		T_Visu.ptrT_ExchgParam^.T_InfoValueCommon.iTotalCountDownCycle:=T_NovRAM.T_Data.T_ProcessImageData.T_AutoGeometryPara.iCycleGeometry;
		T_Visu.ptrT_ExchgParam^.T_InfoValueCommon.iTotalCountDownPlungeCycle:=T_Station.T_WorkTool.iTotalCountDownPlungeCycle;
		T_Visu.ptrT_ExchgParam^.T_InfoValueCommon.iTotalCountDownGrooveCycle:=T_NovRAM.T_Data.T_ProcessImageData.T_AutoGroovePara.iNumberOfGrooves;
		T_Visu.ptrT_ExchgParam^.T_InfoValueCommon.rToolDiameter:=T_NovRAM.T_Data.T_ProcessImageData.T_ProcessPara.rToolDiameterProcess;
		T_Visu.ptrT_ExchgParam^.T_InfoValueCommon.rToolTotalLength:=rToolTotalLength * 10.0;	(* umwandeln von cm in mm *)
		IF (T_Visu.T_PlcParam.dwActualPage = 10) THEN
			IF T_NovRAM.T_Data.T_ProcessImageData.T_AutoGeometryPara.xPlungeActivationGeometry THEN
				T_Visu.ptrT_ExchgParam^.T_InfoValueCommon.rToolTotalLength:=T_Visu.ptrT_ExchgParam^.T_InfoValueCommon.rToolTotalLength + T_NovRAM.T_Data.T_ProcessImageData.T_AutoGeometryPara.rPlungeLengthToolFeedGeometry;
			END_IF;
			IF T_NovRAM.T_Data.T_ProcessImageData.T_AutoGeometryPara.xDisplaceActivationGeometry THEN
				T_Visu.ptrT_ExchgParam^.T_InfoValueCommon.rToolTotalLength:=T_Visu.ptrT_ExchgParam^.T_InfoValueCommon.rToolTotalLength + T_NovRAM.T_Data.T_ProcessImageData.T_AutoGeometryPara.rDisplaceLengthToolFeedGeometry;
			END_IF;
		END_IF;
		IF (T_Visu.T_PlcParam.dwActualPage = 20) THEN
			IF T_NovRAM.T_Data.T_ProcessImageData.T_AutoGroovePara.xPlungeActivationGroove AND NOT(T_NovRAM.T_Data.T_ProcessImageData.T_AutoGroovePara.xBlockGrindFeeder) THEN
				T_Visu.ptrT_ExchgParam^.T_InfoValueCommon.rToolTotalLength:=T_Visu.ptrT_ExchgParam^.T_InfoValueCommon.rToolTotalLength + T_NovRAM.T_Data.T_ProcessImageData.T_AutoGroovePara.rPlungeLengthToolFeedGroove;
			END_IF;
			IF T_NovRAM.T_Data.T_ProcessImageData.T_AutoGroovePara.xDisplaceActivationGroove THEN
				T_Visu.ptrT_ExchgParam^.T_InfoValueCommon.rToolTotalLength:=T_Visu.ptrT_ExchgParam^.T_InfoValueCommon.rToolTotalLength + T_NovRAM.T_Data.T_ProcessImageData.T_AutoGroovePara.rDisplaceLengthToolFeedGroove;
			END_IF;
		END_IF;
	ELSE
		T_Visu.ptrT_ExchgParam^.T_InfoValueCommon.iCountDownCycle:=1;
		T_Visu.ptrT_ExchgParam^.T_InfoValueCommon.iCountDownPlungeCycle:=1;
		T_Visu.ptrT_ExchgParam^.T_InfoValueCommon.iCountDownGrooveCycle:=1;
	END_IF;

(* Tool Geometry Managment *)
	IF (T_Visu.T_PlcParam.dwActualPage = 120) OR (T_Visu.T_PlcParam.dwActualPage = 121) THEN
		FailingEdgeGeometryManagement(CLK:=TRUE);
		RisingEdgeGeometryManagement(CLK:=(T_Visu.T_PlcParam.dwActualPage = 120) OR (T_Visu.T_PlcParam.dwActualPage = 121));
		IF RisingEdgeGeometryManagement.Q THEN
			arSaveToolGeometry:=T_Visu.ptrT_ExchgParam^.T_GeometryCommon.T_Geometry;
		END_IF;
		T_Visu.ptrT_ExchgParam^.T_GeometryCommon.rMinToolDiameter:=T_Visu.ptrT_ExchgParam^.T_StationCommon.T_PrismPara.rToolDiameterMin;
		T_Visu.ptrT_ExchgParam^.T_GeometryCommon.rMaxToolDiameter:=T_Visu.ptrT_ExchgParam^.T_StationCommon.T_PrismPara.rToolDiameterMax;
		T_Visu.ptrT_ExchgParam^.T_GeometryCommon.rMinToolLength:=0.1;
		T_Visu.ptrT_ExchgParam^.T_GeometryCommon.rMaxToolLength:=T_Visu.ptrT_ExchgParam^.T_StationCommon.rConfigMaxToolLength;

		IF (arSaveToolGeometry.arEndDiameter[1] <> T_Visu.ptrT_ExchgParam^.T_GeometryCommon.T_Geometry.arEndDiameter[1]) THEN
			arSaveToolGeometry.arEndDiameter[1]:=T_Visu.ptrT_ExchgParam^.T_GeometryCommon.T_Geometry.arEndDiameter[1];
			arSaveToolGeometry.arStartDiameter[2]:=arSaveToolGeometry.arEndDiameter[1];
			T_Visu.ptrT_ExchgParam^.T_GeometryCommon.T_Geometry.arStartDiameter[2]:=arSaveToolGeometry.arStartDiameter[2];
		END_IF;
		IF (arSaveToolGeometry.arStartDiameter[2] <> T_Visu.ptrT_ExchgParam^.T_GeometryCommon.T_Geometry.arStartDiameter[2]) THEN
			arSaveToolGeometry.arStartDiameter[2]:=T_Visu.ptrT_ExchgParam^.T_GeometryCommon.T_Geometry.arStartDiameter[2];
			arSaveToolGeometry.arEndDiameter[1]:=arSaveToolGeometry.arStartDiameter[2];
			T_Visu.ptrT_ExchgParam^.T_GeometryCommon.T_Geometry.arEndDiameter[1]:=arSaveToolGeometry.arEndDiameter[1];
		END_IF;
		IF (arSaveToolGeometry.arEndDiameter[2] <> T_Visu.ptrT_ExchgParam^.T_GeometryCommon.T_Geometry.arEndDiameter[2]) THEN
			arSaveToolGeometry.arEndDiameter[2]:=T_Visu.ptrT_ExchgParam^.T_GeometryCommon.T_Geometry.arEndDiameter[2];
			arSaveToolGeometry.arStartDiameter[3]:=arSaveToolGeometry.arEndDiameter[2];
			T_Visu.ptrT_ExchgParam^.T_GeometryCommon.T_Geometry.arStartDiameter[3]:=arSaveToolGeometry.arStartDiameter[3];
		END_IF;
		IF (arSaveToolGeometry.arStartDiameter[3] <> T_Visu.ptrT_ExchgParam^.T_GeometryCommon.T_Geometry.arStartDiameter[3]) THEN
			arSaveToolGeometry.arStartDiameter[3]:=T_Visu.ptrT_ExchgParam^.T_GeometryCommon.T_Geometry.arStartDiameter[3];
			arSaveToolGeometry.arEndDiameter[2]:=arSaveToolGeometry.arStartDiameter[3];
			T_Visu.ptrT_ExchgParam^.T_GeometryCommon.T_Geometry.arEndDiameter[2]:=arSaveToolGeometry.arEndDiameter[2];
		END_IF;
		IF (arSaveToolGeometry.arEndDiameter[3] <> T_Visu.ptrT_ExchgParam^.T_GeometryCommon.T_Geometry.arEndDiameter[3]) THEN
			arSaveToolGeometry.arEndDiameter[3]:=T_Visu.ptrT_ExchgParam^.T_GeometryCommon.T_Geometry.arEndDiameter[3];
			arSaveToolGeometry.arStartDiameter[4]:=arSaveToolGeometry.arEndDiameter[3];
			T_Visu.ptrT_ExchgParam^.T_GeometryCommon.T_Geometry.arStartDiameter[4]:=arSaveToolGeometry.arStartDiameter[4];
		END_IF;
		IF (arSaveToolGeometry.arStartDiameter[4] <> T_Visu.ptrT_ExchgParam^.T_GeometryCommon.T_Geometry.arStartDiameter[4]) THEN
			arSaveToolGeometry.arStartDiameter[4]:=T_Visu.ptrT_ExchgParam^.T_GeometryCommon.T_Geometry.arStartDiameter[4];
			arSaveToolGeometry.arEndDiameter[3]:=arSaveToolGeometry.arStartDiameter[4];
			T_Visu.ptrT_ExchgParam^.T_GeometryCommon.T_Geometry.arEndDiameter[3]:=arSaveToolGeometry.arEndDiameter[3];
		END_IF;
(*09.12.2022: SOA	{	 *)
		IF (arSaveToolGeometry.arEndDiameter[4] <> T_Visu.ptrT_ExchgParam^.T_GeometryCommon.T_Geometry.arEndDiameter[4]) THEN
			arSaveToolGeometry.arEndDiameter[4]:=T_Visu.ptrT_ExchgParam^.T_GeometryCommon.T_Geometry.arEndDiameter[4];
			arSaveToolGeometry.arStartDiameter[5]:=arSaveToolGeometry.arEndDiameter[4];
			T_Visu.ptrT_ExchgParam^.T_GeometryCommon.T_Geometry.arStartDiameter[5]:=arSaveToolGeometry.arStartDiameter[5];
		END_IF;
		IF (arSaveToolGeometry.arStartDiameter[5] <> T_Visu.ptrT_ExchgParam^.T_GeometryCommon.T_Geometry.arStartDiameter[5]) THEN
			arSaveToolGeometry.arStartDiameter[5]:=T_Visu.ptrT_ExchgParam^.T_GeometryCommon.T_Geometry.arStartDiameter[5];
			arSaveToolGeometry.arEndDiameter[4]:=arSaveToolGeometry.arStartDiameter[5];
			T_Visu.ptrT_ExchgParam^.T_GeometryCommon.T_Geometry.arEndDiameter[4]:=arSaveToolGeometry.arEndDiameter[4];
		END_IF;
		IF (arSaveToolGeometry.arEndDiameter[5] <> T_Visu.ptrT_ExchgParam^.T_GeometryCommon.T_Geometry.arEndDiameter[5]) THEN
			arSaveToolGeometry.arEndDiameter[5]:=T_Visu.ptrT_ExchgParam^.T_GeometryCommon.T_Geometry.arEndDiameter[5];
			arSaveToolGeometry.arStartDiameter[6]:=arSaveToolGeometry.arEndDiameter[5];
			T_Visu.ptrT_ExchgParam^.T_GeometryCommon.T_Geometry.arStartDiameter[6]:=arSaveToolGeometry.arStartDiameter[6];
		END_IF;
		IF (arSaveToolGeometry.arStartDiameter[6] <> T_Visu.ptrT_ExchgParam^.T_GeometryCommon.T_Geometry.arStartDiameter[6]) THEN
			arSaveToolGeometry.arStartDiameter[6]:=T_Visu.ptrT_ExchgParam^.T_GeometryCommon.T_Geometry.arStartDiameter[6];
			arSaveToolGeometry.arEndDiameter[5]:=arSaveToolGeometry.arStartDiameter[6];
			T_Visu.ptrT_ExchgParam^.T_GeometryCommon.T_Geometry.arEndDiameter[5]:=arSaveToolGeometry.arEndDiameter[5];
		END_IF;
(*09.12.2022: SOA	}	 *)

(*Select Form*)
		FOR ii:=1 TO 6 DO
			IF NOT(T_Visu.ptrT_ExchgParam^.T_GeometryCommon.T_Geometry.axActiveSection[ii]) THEN
				T_Visu.ptrT_ExchgParam^.T_GeometryCommon.abSectionSelectForm[ii]:=0;
			END_IF;
		END_FOR;
		FOR ii:=1 TO 6 DO
			IF (T_Visu.ptrT_ExchgParam^.T_GeometryCommon.T_Geometry.arStartDiameter[ii] = T_Visu.ptrT_ExchgParam^.T_GeometryCommon.T_Geometry.arEndDiameter[ii]) THEN
				IF T_Visu.ptrT_ExchgParam^.T_GeometryCommon.T_Geometry.axActiveSection[ii] THEN
					T_Visu.ptrT_ExchgParam^.T_GeometryCommon.abSectionSelectForm[ii]:=2;
				END_IF;
			END_IF;
		END_FOR;
		FOR ii:=1 TO 6 DO
			IF (T_Visu.ptrT_ExchgParam^.T_GeometryCommon.T_Geometry.arStartDiameter[ii] > T_Visu.ptrT_ExchgParam^.T_GeometryCommon.T_Geometry.arEndDiameter[ii]) THEN
				IF T_Visu.ptrT_ExchgParam^.T_GeometryCommon.T_Geometry.axActiveSection[ii] THEN
					T_Visu.ptrT_ExchgParam^.T_GeometryCommon.abSectionSelectForm[ii]:=3;
				END_IF;
			END_IF;
		END_FOR;
		FOR ii:=1 TO 6 DO
			IF (T_Visu.ptrT_ExchgParam^.T_GeometryCommon.T_Geometry.arStartDiameter[ii] < T_Visu.ptrT_ExchgParam^.T_GeometryCommon.T_Geometry.arEndDiameter[ii]) THEN
				IF T_Visu.ptrT_ExchgParam^.T_GeometryCommon.T_Geometry.axActiveSection[ii] THEN
					T_Visu.ptrT_ExchgParam^.T_GeometryCommon.abSectionSelectForm[ii]:=4;
				END_IF;
			END_IF;
		END_FOR;

 (*Checking for forbidden ToolDiameter - if forbidden: Set Bit in Word *)
	rCalcTotalToolLength:=0.0;
		FOR ii:=1 TO 6 DO
			IF ii>=1 AND ii<=4 THEN
				IF (T_Visu.ptrT_ExchgParam^.T_GeometryCommon.T_Geometry.arStartDiameter[ii] = 0) OR
				     (T_Visu.ptrT_ExchgParam^.T_GeometryCommon.T_Geometry.arStartDiameter[ii] > T_Visu.ptrT_ExchgParam^.T_StationCommon.T_PrismPara.rToolDiameterMax) OR
				     (T_Visu.ptrT_ExchgParam^.T_GeometryCommon.T_Geometry.arStartDiameter[ii] < T_Visu.ptrT_ExchgParam^.T_StationCommon.T_PrismPara.rToolDiameterMin) THEN
					T_Visu.ptrT_ExchgParam^.T_GeometryCommon.wWrongInput:=DWORD_TO_WORD(SETBIT32(T_Visu.ptrT_ExchgParam^.T_GeometryCommon.wWrongInput,INT_TO_SINT(ii-1)));
				ELSE
					T_Visu.ptrT_ExchgParam^.T_GeometryCommon.wWrongInput:=DWORD_TO_WORD(CLEARBIT32(T_Visu.ptrT_ExchgParam^.T_GeometryCommon.wWrongInput,INT_TO_SINT(ii-1)));
				END_IF;
				IF (T_Visu.ptrT_ExchgParam^.T_GeometryCommon.T_Geometry.arEndDiameter[ii] = 0) OR
				     (T_Visu.ptrT_ExchgParam^.T_GeometryCommon.T_Geometry.arEndDiameter[ii] > T_Visu.ptrT_ExchgParam^.T_StationCommon.T_PrismPara.rToolDiameterMax) OR
				     (T_Visu.ptrT_ExchgParam^.T_GeometryCommon.T_Geometry.arEndDiameter[ii] < T_Visu.ptrT_ExchgParam^.T_StationCommon.T_PrismPara.rToolDiameterMin) THEN
					T_Visu.ptrT_ExchgParam^.T_GeometryCommon.wWrongInput:=DWORD_TO_WORD(SETBIT32(T_Visu.ptrT_ExchgParam^.T_GeometryCommon.wWrongInput,INT_TO_SINT(ii+3)));
				ELSE
					T_Visu.ptrT_ExchgParam^.T_GeometryCommon.wWrongInput:=DWORD_TO_WORD(CLEARBIT32(T_Visu.ptrT_ExchgParam^.T_GeometryCommon.wWrongInput,INT_TO_SINT(ii+3)));
				END_IF;
				IF (T_Visu.ptrT_ExchgParam^.T_GeometryCommon.T_Geometry.arSectionPitch[ii] = 0) THEN
					T_Visu.ptrT_ExchgParam^.T_GeometryCommon.wWrongInput:=DWORD_TO_WORD(SETBIT32(T_Visu.ptrT_ExchgParam^.T_GeometryCommon.wWrongInput,INT_TO_SINT(ii+7)));
				ELSE
					T_Visu.ptrT_ExchgParam^.T_GeometryCommon.wWrongInput:=DWORD_TO_WORD(CLEARBIT32(T_Visu.ptrT_ExchgParam^.T_GeometryCommon.wWrongInput,INT_TO_SINT(ii+7)));
				END_IF;
				IF (T_Visu.ptrT_ExchgParam^.T_GeometryCommon.T_Geometry.arSectionLength[ii] = 0) THEN
					T_Visu.ptrT_ExchgParam^.T_GeometryCommon.wWrongInput:=DWORD_TO_WORD(SETBIT32(T_Visu.ptrT_ExchgParam^.T_GeometryCommon.wWrongInput,INT_TO_SINT(ii+11)));
				ELSE
					T_Visu.ptrT_ExchgParam^.T_GeometryCommon.wWrongInput:=DWORD_TO_WORD(CLEARBIT32(T_Visu.ptrT_ExchgParam^.T_GeometryCommon.wWrongInput,INT_TO_SINT(ii+11)));
				END_IF;
 (*09.12.2022: SOA *) (*Definition of second variable = wWrongInput_2*)
			ELSIF  ii>=5 AND ii<=6 THEN
				IF (T_Visu.ptrT_ExchgParam^.T_GeometryCommon.T_Geometry.arSectionPitch[ii] = 0) THEN
					T_Visu.ptrT_ExchgParam^.T_GeometryCommon.wWrongInput_2:=DWORD_TO_WORD(SETBIT32(T_Visu.ptrT_ExchgParam^.T_GeometryCommon.wWrongInput_2,INT_TO_SINT(ii-5)));
				ELSE
					T_Visu.ptrT_ExchgParam^.T_GeometryCommon.wWrongInput_2:=DWORD_TO_WORD(CLEARBIT32(T_Visu.ptrT_ExchgParam^.T_GeometryCommon.wWrongInput_2,INT_TO_SINT(ii-5)));
				END_IF;
				IF (T_Visu.ptrT_ExchgParam^.T_GeometryCommon.T_Geometry.arSectionLength[ii] = 0) THEN
					T_Visu.ptrT_ExchgParam^.T_GeometryCommon.wWrongInput_2:=DWORD_TO_WORD(SETBIT32(T_Visu.ptrT_ExchgParam^.T_GeometryCommon.wWrongInput_2,INT_TO_SINT(ii-1)));
				ELSE
					T_Visu.ptrT_ExchgParam^.T_GeometryCommon.wWrongInput_2:=DWORD_TO_WORD(CLEARBIT32(T_Visu.ptrT_ExchgParam^.T_GeometryCommon.wWrongInput_2,INT_TO_SINT(ii-1)));
				END_IF;
			END_IF;

			IF T_Visu.ptrT_ExchgParam^.T_GeometryCommon.T_Geometry.axActiveSection[ii] THEN
				rCalcTotalToolLength:=rCalcTotalToolLength + T_Visu.ptrT_ExchgParam^.T_GeometryCommon.T_Geometry.arSectionLength[ii];
			END_IF;
		END_FOR;

 (*Checking  every Section for active Bits, changing "SelectForm" if active *)
		IF (rCalcTotalToolLength > T_Visu.ptrT_ExchgParam^.T_StationCommon.rConfigMaxToolLength) AND ((T_Visu.ptrT_ExchgParam^.T_GeometryCommon.wWrongInput AND 16#F000) = 0) THEN
			T_Visu.ptrT_ExchgParam^.T_GeometryCommon.wWrongInput:=T_Visu.ptrT_ExchgParam^.T_GeometryCommon.wWrongInput OR 16#F000;
		END_IF;
		IF T_Visu.ptrT_ExchgParam^.T_GeometryCommon.T_Geometry.axActiveSection[1] THEN
			IF ((T_Visu.ptrT_ExchgParam^.T_GeometryCommon.wWrongInput AND 16#1111) <> 0) THEN
				T_Visu.ptrT_ExchgParam^.T_GeometryCommon.abSectionSelectForm[1]:=5;
			END_IF;
		END_IF;
		IF T_Visu.ptrT_ExchgParam^.T_GeometryCommon.T_Geometry.axActiveSection[2] THEN
			IF ((T_Visu.ptrT_ExchgParam^.T_GeometryCommon.wWrongInput AND 16#2222) <> 0) THEN
				T_Visu.ptrT_ExchgParam^.T_GeometryCommon.abSectionSelectForm[2]:=5;
			END_IF;
		END_IF;
		IF T_Visu.ptrT_ExchgParam^.T_GeometryCommon.T_Geometry.axActiveSection[3] THEN
			IF ((T_Visu.ptrT_ExchgParam^.T_GeometryCommon.wWrongInput AND 16#4444) <> 0) THEN
				T_Visu.ptrT_ExchgParam^.T_GeometryCommon.abSectionSelectForm[3]:=5;
			END_IF;
		END_IF;
		IF T_Visu.ptrT_ExchgParam^.T_GeometryCommon.T_Geometry.axActiveSection[4] THEN
			IF ((T_Visu.ptrT_ExchgParam^.T_GeometryCommon.wWrongInput AND 16#8888) <> 0) THEN
				T_Visu.ptrT_ExchgParam^.T_GeometryCommon.abSectionSelectForm[4]:=5;
			END_IF;
		END_IF;
(*09.12.2022: SOA	}	 *)
		IF T_Visu.ptrT_ExchgParam^.T_GeometryCommon.T_Geometry.axActiveSection[5] THEN
			IF ((T_Visu.ptrT_ExchgParam^.T_GeometryCommon.wWrongInput_2 AND 16#1111) <> 0) THEN
				T_Visu.ptrT_ExchgParam^.T_GeometryCommon.abSectionSelectForm[5]:=5;
			END_IF;
		END_IF;
		IF T_Visu.ptrT_ExchgParam^.T_GeometryCommon.T_Geometry.axActiveSection[6] THEN
			IF ((T_Visu.ptrT_ExchgParam^.T_GeometryCommon.wWrongInput_2 AND 16#2222) <> 0) THEN
				T_Visu.ptrT_ExchgParam^.T_GeometryCommon.abSectionSelectForm[6]:=5;
			END_IF;
		END_IF;
(*09.12.2022: SOA	}	 *)

	ELSE
		RisingEdgeGeometryManagement(CLK:=FALSE);
		FailingEdgeGeometryManagement(CLK:=FALSE);
		(*If the page changes, then copy again the settled value *)
		IF FailingEdgeGeometryManagement.Q THEN
			T_Visu.ptrT_ExchgParam^.T_GeometryCommon.T_Geometry:=T_NovRAM.T_Data.T_ProcessImageData.T_GeometryPara;
		END_IF;
	END_IF;

(* Monitoring Tool Geometry and Tool Calibration calculation Parameter *)
	T_Station.T_WorkTool.iBaseGearDivider:=15000;
	T_Station.T_WorkTool.rPrismaFactor:=T_NovRAM.T_Data.T_ProcessImageData.T_PrismPara.rPrismaFactor;
	T_Station.T_WorkTool.rGrindFeederScaleFactor:=T_Station.THardware.TAxisGrindFeeder.T_CtrleSingle.lrScaleFactor;
	T_Station.T_WorkTool.rToolFeederGearRatio:=T_Station.THardware.TAxisToolFeeder.T_CtrleSingle.lrGearRatio;
	T_Station.T_WorkTool.rToolFeederScaleFactor:=T_Station.THardware.TAxisToolFeeder.T_CtrleSingle.lrScaleFactor;
	T_Station.T_WorkTool.rToolRightGearRatio:=T_Station.THardware.TAxisToolRight.T_CtrleSingle.lrGearRatio;
	IF (T_Visu.T_PlcParam.dwActualPage = 10) OR (T_Visu.T_PlcParam.dwActualPage = 20) THEN
		IF (T_Visu.T_PlcParam.dwActualPage = 10) THEN
			iAutoProcess:=1;
			rToolRotationSpeed:=T_NovRAM.T_Data.T_ProcessImageData.T_AutoGeometryPara.rSpeedToolRotationGeometry;
			T_Station.T_WorkTool.rPlungeSpeedGrindFeed:=T_NovRAM.T_Data.T_ProcessImageData.T_AutoGeometryPara.rPlungeSpeedGrindFeedGeometry;
			T_Station.T_WorkTool.rDisplaceSpeedGrindFeed:=T_NovRAM.T_Data.T_ProcessImageData.T_AutoGeometryPara.rDisplaceSpeedGrindFeedGeometry;
		END_IF;
		IF (T_Visu.T_PlcParam.dwActualPage = 20) THEN
			iAutoProcess:=2;
			rToolRotationSpeed:=T_NovRAM.T_Data.T_ProcessImageData.T_AutoGroovePara.rSpeedToolRotationGroove;
			T_Station.T_WorkTool.rPlungeSpeedGrindFeed:=T_NovRAM.T_Data.T_ProcessImageData.T_AutoGroovePara.rPlungeSpeedGrindFeedGroove;
			T_Station.T_WorkTool.rDisplaceSpeedGrindFeed:=T_NovRAM.T_Data.T_ProcessImageData.T_AutoGroovePara.rDisplaceSpeedGrindFeedGroove;
		END_IF;
	ELSE
		iAutoProcess:=0;
	END_IF;
	IF (((T_Visu.T_PlcParam.dwActualPage = 10) OR (T_Visu.T_PlcParam.dwActualPage = 20) OR (T_Visu.T_PlcParam.dwActualPage = 110)) OR xCalcAgainProcTime) AND T_Visu.T_CtrleVisu.xDone THEN
		IF NOT(xCalcFirstTime) OR xCalcAgainProcTime THEN
			xCalcFirstTime:=TRUE;
			FBCalcProcessTime(	T_Geometry:=T_NovRAM.T_Data.T_ProcessImageData.T_GeometryPara,
								T_AutoGeometryPara:=T_NovRAM.T_Data.T_ProcessImageData.T_AutoGeometryPara,
								T_CalibrationPara:=T_NovRAM.T_Data.T_ProcessImageData.T_CalibrationPara,
								T_AutoGroovePara:=T_NovRAM.T_Data.T_ProcessImageData.T_AutoGroovePara,
								T_ProcessPara:=T_NovRAM.T_Data.T_ProcessImageData.T_ProcessPara,
								rToolRotationSpeed:=rToolRotationSpeed,
								rToolDiameter:=T_NovRAM.T_Data.T_ProcessImageData.T_ProcessPara.rToolDiameterProcess,
								rToolDiameterWithOffset:=	T_NovRAM.T_Data.T_ProcessImageData.T_ProcessPara.rToolDiameterProcess +
														T_NovRAM.T_Data.T_ProcessImageData.T_ProcessPara.rOffsetBeforeToolDiaGrindFeedProcess,
								iAutoProcess:=iAutoProcess,
								xMicroRodActive:=xMicroRodActive,
								T_WorkTool:=T_Station.T_WorkTool);
		END_IF;
		xCalcAgainProcTime:=FALSE;
		rAutoTimeTotal:=FBCalcProcessTime.rProcessTime;
		T_Visu.ptrT_ExchgParam^.T_InfoValueCommon.tAutoTimeTotal:=REAL_TO_TIME(rAutoTimeTotal * 1000.0);
	ELSE
		xCalcFirstTime:=FALSE;
	END_IF;
	IF T_Process.xEnd OR T_Process.xError THEN
		T_Visu.ptrT_ExchgParam^.T_InfoValueCommon.tAutoTimeLeft:=T_Visu.ptrT_ExchgParam^.T_InfoValueCommon.tAutoTimeTotal;
		T_Visu.ptrT_ExchgParam^.T_InfoValueCommon.bProgressbarAutoGeometry:=0;
		T_Visu.ptrT_ExchgParam^.T_InfoValueCommon.bProgressbarAutoGroove:=0;
		T_Visu.ptrT_ExchgParam^.T_InfoValueCommon.bProgressbarToolCalibration:=0;
	END_IF;

(* Monitoring ToolCalibration *)
	IF (T_Visu.T_PlcParam.dwActualPage = 110) THEN
		T_Visu.ptrT_ExchgParam^.T_InfoValueCommon.rToolLengthCalibration:=T_NovRAM.T_Data.T_ProcessImageData.T_CalibrationPara.rToolLengthCylinderPartCalib;
		T_Visu.ptrT_ExchgParam^.T_InfoValueCommon.rToolDiameter:=T_NovRAM.T_Data.T_ProcessImageData.T_ProcessPara.rToolDiameterProcess;
		T_Visu.ptrT_ExchgParam^.T_InfoValueCommon.rPitchCalibration:=T_NovRAM.T_Data.T_ProcessImageData.T_CalibrationPara.rPitchCalib;
	END_IF;

(* Monitoring Correction Tool Diameter *)
	IF (T_Visu.T_PlcParam.dwActualPage = 420) OR (T_Visu.T_PlcParam.dwActualPage = 11) OR (T_Visu.T_PlcParam.dwActualPage = 21) THEN
		RisingEdgeToolDiameter(CLK:=(T_Visu.T_PlcParam.dwActualPage = 420) OR (T_Visu.T_PlcParam.dwActualPage = 11) OR (T_Visu.T_PlcParam.dwActualPage = 21));
		IF RisingEdgeToolDiameter.Q THEN
			T_Visu.ptrT_ExchgParam^.T_InfoValueCommon.rCorrectionToolDiameter:=0.0;
			T_Visu.ptrT_ExchgParam^.T_InfoValueCommon.xKeyPadActivation:=FALSE;
		END_IF;
		IF (T_Visu.ptrT_ExchgParam^.T_InfoValueCommon.rCorrectionToolDiameter = 0) THEN
			T_Visu.ptrT_ExchgParam^.T_StationCommon.bStateToolDiameter:=1;
		END_IF;
		IF (T_Visu.ptrT_ExchgParam^.T_InfoValueCommon.rCorrectionToolDiameter > 0) THEN
			T_Visu.ptrT_ExchgParam^.T_StationCommon.bStateToolDiameter:=3;
		END_IF;
		IF (T_Visu.ptrT_ExchgParam^.T_InfoValueCommon.rCorrectionToolDiameter < 0) THEN
			T_Visu.ptrT_ExchgParam^.T_StationCommon.bStateToolDiameter:=2;
		END_IF;
	ELSE
		RisingEdgeToolDiameter(CLK:=FALSE);
	END_IF

(* Monitoring TeachIn Tool Rotation *)
	IF (T_Visu.T_PlcParam.dwActualPage = 210) THEN
		IF xToolRotationMasterSlave THEN
			T_Visu.ptrT_ExchgParam^.T_TeachIn.iSelectAxisToolRotation:=1;	(* Force Selection by choice of MasterSlave to the ToolLeft TouchButton *)
		END_IF;
		IF (T_Visu.ptrT_ExchgParam^.T_SafetyCtrl.bStateTeachInToolLeft = 2) OR (T_Visu.ptrT_ExchgParam^.T_SafetyCtrl.bStateTeachInToolCenter = 2) OR
		     (T_Visu.ptrT_ExchgParam^.T_SafetyCtrl.bStateTeachInToolRight = 2) THEN
			T_Visu.ptrT_ExchgParam^.T_TeachIn.iSelectAxisToolRotation:=iSelectAxisToolRotation;	(* Force Selection by active movement *)
		END_IF;
		IF (T_Visu.ptrT_ExchgParam^.T_TeachIn.iSelectAxisToolRotation <> iSelectAxisToolRotation) THEN
			iSelectAxisToolRotation:=T_Visu.ptrT_ExchgParam^.T_TeachIn.iSelectAxisToolRotation;
		END_IF;
	END_IF;
	IF (T_Visu.T_PlcParam.dwActualPage <> 210) AND xToolRotationMasterSlave THEN
		xToolRotationMasterSlave:=FALSE;
		IF xMicroRodActive THEN
			IF T_Station.THardware.TAxisToolCenter.T_CtrleSingle.xSlave AND T_Station.THardware.TAxisToolCenter.T_CtrleSingle.xDone THEN
				T_Station.THardware.TAxisToolCenter.T_CtrleSingle.iFunction:=25;
				T_Station.THardware.TAxisToolCenter.T_CtrleSingle.xExecute:=TRUE;
			END_IF;
		END_IF;
		IF T_Station.THardware.TAxisToolRight.T_CtrleSingle.xSlave AND T_Station.THardware.TAxisToolRight.T_CtrleSingle.xDone THEN
			T_Station.THardware.TAxisToolRight.T_CtrleSingle.iFunction:=25;
			T_Station.THardware.TAxisToolRight.T_CtrleSingle.xExecute:=TRUE;
		END_IF;
		IF NOT(xMicroRodActive) THEN
			IF T_Station.THardware.TAxisToolFeeder.T_CtrleSingle.xSlave AND T_Station.THardware.TAxisToolFeeder.T_CtrleSingle.xDone THEN
				T_Station.THardware.TAxisToolFeeder.T_CtrleSingle.iFunction:=25;
				T_Station.THardware.TAxisToolFeeder.T_CtrleSingle.xExecute:=TRUE;
			END_IF;
		END_IF;
	END_IF;

(* Monitoring Prisma *)
	IF (T_Visu.T_PlcParam.dwActualPage = 430) THEN
		FailingEdgePrisma(CLK:=TRUE);
		RisingEdgePrisma(CLK:=(T_Visu.T_PlcParam.dwActualPage = 430));
		IF RisingEdgePrisma.Q THEN
		(* 0= 3 value prisma, 1 = 3 value prisma input para, 2 = 2 value prisma, 3 = 2 value prisma input para *)
			IF (T_Visu.ptrT_ExchgParam^.T_StationCommon.T_PrismPara.bStateInputPrisma = 1) THEN
				T_Visu.ptrT_ExchgParam^.T_StationCommon.T_PrismPara.bStateInputPrisma:=0;
			END_IF;
			IF (T_Visu.ptrT_ExchgParam^.T_StationCommon.T_PrismPara.bStateInputPrisma = 3) THEN
				T_Visu.ptrT_ExchgParam^.T_StationCommon.T_PrismPara.bStateInputPrisma:=2;
			END_IF;
		END_IF;
	ELSE
		RisingEdgePrisma(CLK:=FALSE);
		FailingEdgePrisma(CLK:=FALSE);
		(*If the page changes, then copy again the settled value *)
		IF FailingEdgePrisma.Q THEN
			T_Visu.ptrT_ExchgParam^.T_StationCommon.T_PrismPara:=T_NovRAM.T_Data.T_ProcessImageData.T_PrismPara;
		END_IF;
	END_IF

(* Tmp timer *)
	TimerONTmp(IN:=TRUE);

(************************************************************************************************************************************************************************)
(***************                                          start of the management for call a function of the visualisation interface                                           ********************)
(************************************************************************************************************************************************************************)
(* waiting for executing action *)
	(* ...monitor Key panel "Enter" *)
	RisingEdgeKeyPanel_Enter(CLK:=T_Visu.ptrT_ExchgParam^.T_Visu.xKey_Enter);
	(* ...monitor Key panel "Esc" *)
	RisingEdgeKeyPanel_Esc(CLK:=T_Visu.ptrT_ExchgParam^.T_Visu.xKey_Escape);
	IF RisingEdgeKeyPanel_Esc.Q THEN tTimeOutAction:=TimerAction.ET; END_IF
	(*... not ready *)
	TimerNotReady(IN:=FALSE, PT:=T#2s);
	T_Visu.T_CtrleAction.xNotReady:=TimerNotReady.Q;

(* ...message *)
	RisingEdgeActionNotReady(CLK:=T_Visu.T_CtrleAction.xNotReady);
	IF RisingEdgeActionNotReady.Q AND T_Visu.ptrT_ExchgParam^.T_Visu.T_Message.iState < 200 THEN
		T_Visu.ptrT_ExchgParam^.T_Visu.T_Message.iState:=101; END_IF
	(* Release 'Not ready' action control structure *)
	FallingEdgeActionNotReady(CLK:=T_Visu.T_CtrleAction.xNotReady);
	IF FallingEdgeActionNotReady.Q THEN
		IF (T_Visu.ptrT_ExchgParam^.T_Visu.T_Message.iState =101) THEN
			T_Visu.ptrT_ExchgParam^.T_Visu.T_Message.iState:=0;
		END_IF;
		T_Visu.T_CtrleAction.xExecute:=FALSE;
		T_Visu.T_CtrleAction.xDone:=TRUE;
		T_Visu.T_CtrleAction.xErr:=FALSE;
		T_Visu.T_CtrleAction.udiErrorID:=0;
		iStepAction:=1;
		(*
		iStepActionRef:=1;
		iStepActionNovRam:=1;
		*)
		xStepActionDone:=FALSE;
		TimerAction(IN:=FALSE);
	END_IF
	(* ...done *)
	RisingEdgeActionDone(CLK:=T_Visu.T_CtrleAction.xDone);
	IF RisingEdgeActionDone.Q THEN
		(* disable mask stop action *)
		(*wStopActionMaskBtPanelRight:=16#0;*)
		(*xWaitingReleaseStopBtPanel:=FALSE;*)
		IF T_Visu.T_CtrleAction.iFunction > 100
		    AND (T_Visu.ptrT_ExchgParam^.T_Visu.T_Message.iState = 0 OR (T_Visu.ptrT_ExchgParam^.T_Visu.T_Message.iState  > 100 AND T_Visu.ptrT_ExchgParam^.T_Visu.T_Message.iState < 200)) THEN
			IF NOT TimerAction.Q AND NOT FallingEdgeActionNotReady.Q THEN
				IF NOT(xBlockConfirmMessage) THEN
					(* call confirmation message *)
					T_Visu.ptrT_ExchgParam^.T_Visu.T_Message.iState
						:=iFctReturnConfMessage(iNumAction:=T_Visu.T_CtrleAction.iFunction);
				ELSE
					xBlockConfirmMessage:=FALSE;
				END_IF;
			(* call cancelled message *)
			ELSE T_Visu.ptrT_ExchgParam^.T_Visu.T_Message.iState:=5; END_IF
		END_IF
	END_IF
	(* ...error *)
	RisingEdgeActionError(CLK:=T_Visu.T_CtrleAction.xErr);
	IF RisingEdgeActionError.Q THEN
	(* call function bloc action error *)
		(*fbQvisError(	udiActionError:=T_Visu.T_CtrleAction.udiErrorID,
					T_Message:=T_Visu.ptrT_ExchgParam^.T_Visu.T_Message);*)
		(* Init. variable *)
		T_Visu.T_CtrleAction.xExecute:=FALSE;
		T_Visu.T_CtrleAction.xDone:=TRUE;
		T_Visu.T_CtrleAction.xErr:=FALSE;
		T_Visu.T_CtrleAction.xNotReady:=FALSE;
		T_Visu.T_CtrleAction.udiErrorID:=0;
		iStepAction:=1;
		(*
		iStepActionRef:=1;
		iStepActionNovRam:=1;
		*)
		xStepActionDone:=FALSE;
	END_IF
	(* ...reset *)
	RisingEdgeResetAction(CLK:=T_Visu.T_CtrleAction.xReset);
	IF RisingEdgeResetAction.Q THEN
		(* Init. variable *)
		T_Visu.T_CtrleAction.xExecute:=FALSE;
		T_Visu.T_CtrleAction.xDone:=TRUE;
		T_Visu.T_CtrleAction.xErr:=FALSE;
		T_Visu.T_CtrleAction.xNotReady:=FALSE;
		T_Visu.T_CtrleAction.udiErrorID:=0;
		iStepAction:=1;
		(*
		iStepActionRef:=1;
		iStepActionNovRam:=1;
		*)
		xStepActionDone:=FALSE;
		TimerAction(IN:=FALSE);
		(* Release reset *)
		T_Visu.T_CtrleAction.xReset:=FALSE;
	END_IF

	(* Execute Function *)
	RisingEdgeExecuteAction(CLK:=T_Visu.T_CtrleAction.xExecute);
	IF RisingEdgeExecuteAction.Q THEN
		(* confirm action execution *)
		T_Visu.T_CtrleAction.xExecute:=FALSE;
		CASE T_Visu.T_CtrleAction.iFunction OF
			(* Set parameter page *)
			3:	xSetParameterPage:=TRUE;
				tTimeOutAction:=T#3s;
			(* Change Page Button Panel Left *)
			6:	xBtPanelLeftChangePage:=TRUE;
				tTimeOutAction:=T#3s;
	(*SOA 13.01.2023  { *)
			(* Change Page Button Panel Right *)
			7:	xBtPanelRightChangePage:=TRUE;
				tTimeOutAction:=T#3s;
	(*SOA 13.01.2023  } *)
			(* next page vertical *)
			12:	xNextPageVertical:=TRUE;
				tTimeOutAction:=T#3s;
			(* Delete error List *)
			20:	xDeleteErrorList:=TRUE;
				tTimeOutAction:=T#3s;
			(* Reset error *)
			99:	xResetError:=TRUE;
				tTimeOutAction:=T#3s;
			(* Open Overlay for input measured tool diameter *)
			101:	xOverlayMeasureToolDia:=TRUE;
				tTimeOutAction:=T#9999s;
			(* Plunge On/Off *)
			102:	xPlungeActivation:=TRUE;
				tTimeOutAction:=T#3s;
			(* Displace On/Off *)
			103:	xDisplaceActivation:=TRUE;
				tTimeOutAction:=T#3s;
			(* AutoGroove-->Block GrindFeeder On/Off *)
			104:	xBlockGrindFeederActivation:=TRUE;
				tTimeOutAction:=T#3s;
			(* AutoGroove-->ToolFeeder move to StartPos *)
			105:	xToolFeederMoveStartPos:=TRUE;
				tTimeOutAction:=T#3s;
			(* AutoGeometry and AutoGroove-->Switch On/Off all Axis Power *)
			106:	xToggleAllAxisPower:=TRUE;
				tTimeOutAction:=T#3s;
			(* AutoGeometry and AutoGroove-->ToolFeeder move to LoadPos *)
			107:	xToolFeederMoveLoadPos:=TRUE;
				tTimeOutAction:=T#3s;
(*08.07.2014: KFS	{	*)
			(* AutoGeometry -->WarmUp On/OFF *)
			108:	xWarmUp:=TRUE;
				tTimeOutAction:=T#3s;
(*08.07.2014: KFS	}	*)
			(* Correction Tool Diameter + *)
			110:	xCorrectionToolDiameterAdd:=TRUE;
				tTimeOutAction:=T#3s;
			(* Correction Tool Diameter ++ *)
			111:	xCorrectionToolDiameterAddMore:=TRUE;
				tTimeOutAction:=T#3s;
			(* Correction Tool Diameter - *)
			112:	xCorrectionToolDiameterSub:=TRUE;
				tTimeOutAction:=T#3s;
			(* Correction Tool Diameter -- *)
			113:	xCorrectionToolDiameterSubMore:=TRUE;
				tTimeOutAction:=T#3s;
			(* Reset Tool Diameter Correction *)
			114:	xResetToolDiameterCorrection:=TRUE;
				tTimeOutAction:=T#3s;
			(* Keypad Activation *)
			115: xKeyPadActivation:=TRUE;
				tTimeOutAction:=T#3s;
			(* Function Correction Tool Diameter *)
			116:	xFctCorrectionToolDiameter:=TRUE;
				tTimeOutAction:=T#3s;
			(* Select Prisma 1 or 2 Input *)
			120:	xSelectPrisma:=TRUE;
				tTimeOutAction:=T#3s;
			(* Set calculated ToolRotation Torque *)
			130:	xSetCalculToolRotTorque:=TRUE;
				tTimeOutAction:=T#3s;
			(* Reset calculated ToolRotation Torque *)
			131:	xResetCalculToolRotTorque:=TRUE;
				tTimeOutAction:=T#3s;
			(* Open Overlay for input the correction of the position of the GrindFeeder *)
			132:	xOverlayGrindFeedSetPlung:=TRUE;
				tTimeOutAction:=T#9999s;
	(*SOA 13.01.2023  { *)
			173:	xConfirmStartWarmUp:=TRUE;
				tTimeOutAction:=T#3s;
			(* Stop Warmupl  *)
			175: 	xStopWarmup:=TRUE;
				tTimeOutAction:=T#3s;
	(*SOA 13.01.2023  } *)
			(* Activation Section 1 *) (*
			201: (* 13.10.2010 KFS 	{ 	*)
				(*	xActivationSection1:=TRUE;
					tTimeOutAction:=T#3s;			*)
				(* 13.10.2010 KFS   }	 *) *)
			(* Activation Section 2 *)
			202:	xActivationSection2:=TRUE;
				tTimeOutAction:=T#3s;
			(* Activation Section 3 *)
			203:	xActivationSection3:=TRUE;
				tTimeOutAction:=T#3s;
			(* Activation Section 4 *)
			204:	xActivationSection4:=TRUE;
				tTimeOutAction:=T#3s;
			(* Set pitch equal *)
			205:	xSetPitchEqual:=TRUE;
				tTimeOutAction:=T#3s;
	(* 13.10.2022 SOA*)
			(* Activation Section 5 *)
			206:	xActivationSection5:=TRUE;
				tTimeOutAction:=T#3s;
			(* Activation Section 6 *)
			207:	xActivationSection6:=TRUE;
				tTimeOutAction:=T#3s;
	(* 13.10.2022 SOA*)
			(* TeachIN page *)
			301..399:	(* set pointer, default pointer axis slide *)
					ptrTeachINAxis:=ADR(T_Station.THardware.TAxisToolLeft);
					iSelectedAxis:=1;
					IF (T_Visu.T_PlcParam.dwActualPage = 210) THEN
						xSlowFast:=T_Visu.ptrT_ExchgParam^.T_TeachIn.xSlowFastToolRotation;
						IF (T_Visu.ptrT_ExchgParam^.T_TeachIn.iSelectAxisToolRotation = 1) THEN
							iSelectedAxis:=1;
							TParaAxisTeachIN:=T_Visu.ptrT_ExchgParam^.T_TeachIn.TParam_ToolLeft:=T_NovRam.T_Data.T_Standard.T_TeachINToolLeft;
							ptrTeachINAxis:=ADR(T_Station.THardware.TAxisToolLeft);
						END_IF;
						IF (T_Visu.ptrT_ExchgParam^.T_TeachIn.iSelectAxisToolRotation = 2) THEN
							iSelectedAxis:=2;
							TParaAxisTeachIN:=T_Visu.ptrT_ExchgParam^.T_TeachIn.TParam_ToolCenter:=T_NovRam.T_Data.T_Standard.T_TeachINToolCenter;
							ptrTeachINAxis:=ADR(T_Station.THardware.TAxisToolCenter);
						END_IF;
						IF (T_Visu.ptrT_ExchgParam^.T_TeachIn.iSelectAxisToolRotation = 3) THEN
							iSelectedAxis:=3;
							TParaAxisTeachIN:=T_Visu.ptrT_ExchgParam^.T_TeachIn.TParam_ToolRight:=T_NovRam.T_Data.T_Standard.T_TeachINToolRight;
							ptrTeachINAxis:=ADR(T_Station.THardware.TAxisToolRight);
						END_IF;
					END_IF;
					IF (T_Visu.T_PlcParam.dwActualPage = 30) OR (T_Visu.T_PlcParam.dwActualPage = 310) OR (T_Visu.T_PlcParam.dwActualPage = 320) OR (T_Visu.T_PlcParam.dwActualPage = 330) THEN
						iSelectedAxis:=4;
						xSlowFast:=T_Visu.ptrT_ExchgParam^.T_TeachIn.xSlowFastToolFeed;
						TParaAxisTeachIN:=T_Visu.ptrT_ExchgParam^.T_TeachIn.TParam_ToolFeeder:=T_NovRam.T_Data.T_Standard.T_TeachINToolFeeder;
						ptrTeachINAxis:=ADR(T_Station.THardware.TAxisToolFeeder);
					END_IF;
					IF (T_Visu.T_PlcParam.dwActualPage = 410) THEN
						iSelectedAxis:=5;
						xSlowFast:=T_Visu.ptrT_ExchgParam^.T_TeachIn.xSlowFastGrindFeeder;
						TParaAxisTeachIN:=T_Visu.ptrT_ExchgParam^.T_TeachIn.TParam_GrindFeeder:=T_NovRam.T_Data.T_Standard.T_TeachINGrindFeeder;
						ptrTeachINAxis:=ADR(T_Station.THardware.TAxisGrindFeeder);
					END_IF;
					CASE T_Visu.T_CtrleAction.iFunction OF
					(* Stop axis movement *)
					301:	xStopAxis:=TRUE;
						tTimeOutAction:=T#4s;
					(* Move Axis Absolut *)
					305:	IF (iSelectedAxis = 4) THEN
							IF xMicroRodActive THEN
								IF (T_Visu.ptrT_ExchgParam^.T_TeachIn.iSaveToolFeederPos = 0) THEN
									ptrTeachINAxis^.T_CtrleSingle.lrPosition:=T_Visu.ptrT_ExchgParam^.T_StationCommon.rNewToolFeederPosition;
								END_IF;
								IF (T_Visu.ptrT_ExchgParam^.T_TeachIn.iSaveToolFeederPos = 1) THEN
									ptrTeachINAxis^.T_CtrleSingle.lrPosition:=T_NovRam.T_Data.T_ProcessImageData.T_ProcessPara.rStartPosToolFeedAuto;
								END_IF;
								IF (T_Visu.ptrT_ExchgParam^.T_TeachIn.iSaveToolFeederPos = 2) THEN
									ptrTeachINAxis^.T_CtrleSingle.lrPosition:=T_NovRam.T_Data.T_ProcessImageData.T_CalibrationPara.rStartPosToolFeedCalib;
								END_IF;
								IF (T_Visu.ptrT_ExchgParam^.T_TeachIn.iSaveToolFeederPos = 3) THEN
									ptrTeachINAxis^.T_CtrleSingle.lrPosition:=T_NovRam.T_Data.T_ProcessImageData.T_CalibrationPara.rMeasurePosToolFeedCalib;
								END_IF;
								IF (T_Visu.ptrT_ExchgParam^.T_TeachIn.iSaveToolFeederPos = 4) THEN
									ptrTeachINAxis^.T_CtrleSingle.lrPosition:=T_NovRam.T_Data.T_Standard.T_AxisPosition.rLoadPosToolFeedAuto;
								END_IF;
								ptrTeachINAxis^.T_CtrleSingle.lrVelocity:=TParaAxisTeachIN.rPositionSpeed;
								xMoveAbsPosition:=TRUE;
							END_IF;
							IF NOT(xMicroRodActive) THEN
								ptrTeachINAxis^.T_CtrleSingle.lrDistance:=T_Visu.ptrT_ExchgParam^.T_StationCommon.rNewToolFeederPosition;
								ptrTeachINAxis^.T_CtrleSingle.lrVelocity:=TParaAxisTeachIN.rPositionSpeed;
								xMoveRelPosition:=TRUE;
							END_IF;
						END_IF;
						IF (iSelectedAxis = 5) THEN
							IF (T_Visu.ptrT_ExchgParam^.T_TeachIn.iSaveGrindFeederPos = 0) THEN
								ptrTeachINAxis^.T_CtrleSingle.lrPosition:=T_Visu.ptrT_ExchgParam^.T_StationCommon.rNewGrindFeederPosition;
							END_IF;
							IF (T_Visu.ptrT_ExchgParam^.T_TeachIn.iSaveGrindFeederPos = 1) THEN
								ptrTeachINAxis^.T_CtrleSingle.lrPosition:=T_NovRam.T_Data.T_ProcessImageData.T_ProcessPara.rToolDiameterProcess;
							END_IF;
							IF (T_Visu.ptrT_ExchgParam^.T_TeachIn.iSaveGrindFeederPos = 2) THEN
								ptrTeachINAxis^.T_CtrleSingle.lrPosition:=	T_NovRam.T_Data.T_ProcessImageData.T_ProcessPara.rToolDiameterProcess +
																	T_NovRam.T_Data.T_ProcessImageData.T_ProcessPara.rSecurityPosGrindFeedProcess;
							END_IF;
							IF (T_Visu.ptrT_ExchgParam^.T_TeachIn.iSaveGrindFeederPos = 3) THEN
								ptrTeachINAxis^.T_CtrleSingle.lrPosition:=T_NovRam.T_Data.T_ProcessImageData.T_PrismPara.rToolDiameterMin;;
							END_IF;
							IF (T_Visu.ptrT_ExchgParam^.T_TeachIn.iSaveGrindFeederPos = 4) THEN
								ptrTeachINAxis^.T_CtrleSingle.lrPosition:=T_NovRam.T_Data.T_ProcessImageData.T_PrismPara.rToolDiameterMax + T_NovRam.T_Data.T_Standard.T_TeachINGrindFeeder.rOffsetSWPosEndSwitch;
							END_IF;
							ptrTeachINAxis^.T_CtrleSingle.lrVelocity:=TParaAxisTeachIN.rPositionSpeed;
							xMoveAbsPosition:=TRUE;
						END_IF;
						tTimeOutAction:=T#999s;
					(* Move Inc Slow/Fast Pos *)
					310..311: IF NOT(xSlowFast) THEN
								ptrTeachINAxis^.T_CtrleSingle.lrDistance:=TParaAxisTeachIN.rIncSlow;
								ptrTeachINAxis^.T_CtrleSingle.lrVelocity:=TParaAxisTeachIN.rVelSlow;
							ELSE
								ptrTeachINAxis^.T_CtrleSingle.lrDistance:=TParaAxisTeachIN.rIncFast;
								ptrTeachINAxis^.T_CtrleSingle.lrVelocity:=TParaAxisTeachIN.rVelFast;
							END_IF
							xMoveRelPosition:=TRUE;
							tTimeOutAction:=T#200s;
					(* Move Inc Slow/Fast Neg *)
					312..313:	IF NOT(xSlowFast) THEN
								ptrTeachINAxis^.T_CtrleSingle.lrDistance:=TParaAxisTeachIN.rIncSlow * -1.0;
								ptrTeachINAxis^.T_CtrleSingle.lrVelocity:=TParaAxisTeachIN.rVelSlow;
							ELSE
								ptrTeachINAxis^.T_CtrleSingle.lrDistance:=TParaAxisTeachIN.rIncFast * -1.0;
								ptrTeachINAxis^.T_CtrleSingle.lrVelocity:=TParaAxisTeachIN.rVelFast;
							END_IF
							xMoveRelPosition:=TRUE;
							tTimeOutAction:=T#200s;
					(* Move Vel Slow/Fast Pos *)
					314..315:	IF NOT(xSlowFast) THEN
								ptrTeachINAxis^.T_CtrleSingle.lrVelocity:=TParaAxisTeachIN.rVelSlow;
							ELSE
								ptrTeachINAxis^.T_CtrleSingle.lrVelocity:=TParaAxisTeachIN.rVelFast;
							END_IF
							xMoveContinousVel:=TRUE;
							tTimeOutAction:=T#200s;
					(* Move Vel Slow/Fast Neg *)
					316..317:	IF NOT(xSlowFast) THEN
								ptrTeachINAxis^.T_CtrleSingle.lrVelocity:=TParaAxisTeachIN.rVelSlow * -1.0;
							ELSE
								ptrTeachINAxis^.T_CtrleSingle.lrVelocity:=TParaAxisTeachIN.rVelFast * -1.0;
							END_IF
							xMoveContinousVel:=TRUE;
							tTimeOutAction:=T#200s;
					(* Move Continuos Velocity *)
					318:		ptrTeachINAxis^.T_CtrleSingle.lrVelocity:=T_Visu.ptrT_ExchgParam^.T_StationCommon.rNewToolRotationSpeed;
							xMoveContinousVel:=TRUE;
							tTimeOutAction:=T#200s;
					(* Switch WireFeed Jog Speed Slow/Fast *)
					320:		IF ((iSelectedAxis = 1) OR (iSelectedAxis = 2) OR (iSelectedAxis = 3)) AND (T_Visu.T_PlcParam.dwActualPage <> 30) THEN
								xSlowFastJogToolRotation:=TRUE;
							END_IF;
							IF (iSelectedAxis = 4) OR (T_Visu.T_PlcParam.dwActualPage = 30) THEN
								xSlowFastJogToolFeeder:=TRUE;
							END_IF;
							IF (iSelectedAxis = 5) AND (T_Visu.T_PlcParam.dwActualPage <> 30) THEN
								xSlowFastJogGrindFeeder:=TRUE;
							END_IF;
							tTimeOutAction:=T#3s;
					(* Switch ToolRotation Master Slave *)
					321:		IF xMicroRodActive THEN
								(* ToolCenter --> Slave of ToolLeft only by MicroRod *)
								T_Station.THardware.TAxisToolCenter.T_CtrleSingle.lrGearDivider:=INT_TO_LREAL(T_Station.T_WorkTool.iBaseGearDivider);
								T_Station.THardware.TAxisToolCenter.T_CtrleSingle.lrGearFactor:=(	INT_TO_LREAL(T_Station.T_WorkTool.iBaseGearDivider) /
																								(T_Station.THardware.TAxisToolLeft.T_CtrleSingle.lrGearRatio /
																								T_Station.THardware.TAxisToolCenter.T_CtrleSingle.lrGearRatio)) * -1.0;

								(* ToolRight --> Slave of ToolLeft by MicroWire or Slave of ToolRight by MicroRod *)
								T_Station.THardware.TAxisToolRight.T_CtrleSingle.lrGearDivider:=INT_TO_LREAL(T_Station.T_WorkTool.iBaseGearDivider);
								T_Station.THardware.TAxisToolRight.T_CtrleSingle.lrGearFactor:=	INT_TO_LREAL(T_Station.T_WorkTool.iBaseGearDivider) /
																								(T_Station.THardware.TAxisToolLeft.T_CtrleSingle.lrGearRatio /
																								T_Station.THardware.TAxisToolRight.T_CtrleSingle.lrGearRatio);
							END_IF;
							IF NOT(xMicroRodActive) THEN
								(* ToolRight --> Slave of ToolRight by MicroWire *)
								T_Station.THardware.TAxisToolFeeder.T_CtrleSingle.lrGearDivider:=INT_TO_LREAL(T_Station.T_WorkTool.iBaseGearDivider);
								T_Station.THardware.TAxisToolFeeder.T_CtrleSingle.lrGearFactor:=	(INT_TO_LREAL(T_Station.T_WorkTool.iBaseGearDivider) /
																							(T_Station.THardware.TAxisToolFeeder.T_CtrleSingle.lrGearRatio /
																							T_Station.THardware.TAxisToolRight.T_CtrleSingle.lrGearRatio)) * -1.0;

								(* ToolRight --> Slave of ToolLeft by MicroWire or Slave of ToolRight by MicroRod *)
								T_Station.THardware.TAxisToolRight.T_CtrleSingle.lrGearDivider:=INT_TO_LREAL(T_Station.T_WorkTool.iBaseGearDivider);
								T_Station.THardware.TAxisToolRight.T_CtrleSingle.lrGearFactor:=	(INT_TO_LREAL(T_Station.T_WorkTool.iBaseGearDivider) /
																								(T_Station.THardware.TAxisToolLeft.T_CtrleSingle.lrGearRatio /
																								T_Station.THardware.TAxisToolRight.T_CtrleSingle.lrGearRatio)) * -1.0;
							END_IF;
							xSwitchMasterSlave:=TRUE;
							tTimeOutAction:=T#3s;
					(* Power axis *)
					322:		xToggleAxisPower:=TRUE;
							tTimeOutAction:=T#3s;
					(* Reset axis *)
					323:		xResetAxis:=TRUE;
							tTimeOutAction:=T#3s;
					(* Reference axis *)
					324:		xReferenceAxis:=TRUE;
							tTimeOutAction:=T#200s;
					(* Teach axis Position *)
					325:		xTeachPosition:=TRUE;
							tTimeOutAction:=T#6s;
					(* Calculate the position between the RefIndex and the RefSensor *)
					326:		xCalcAngleRefIndex:=TRUE;
							tTimeOutAction:=T#200s;
					END_CASE;
			(* Station Function *)
			401..499:	xActivateStationFunction:=TRUE;
					iTmpStationFunctionNr:=T_Visu.T_CtrleAction.iFunction - 400;	(* Select Function Number 1 - 99 *)
					IF (iTmpStationFunctionNr = 20) THEN tTimeOutAction:=T#200s; ELSE tTimeOutAction:=T#3s;END_IF;
			(* Cylinder Function *)
			501..599:	(* set pointer, default pointer CylToolTension *)
					(* 1=CylToolTension, 2=CylToolLeftActive, 3=CylToolRightActive, 4=CylToolCenter,5=CylToolPrismaLeftActive, 6=CylToolPrismaRightActive *)
					ptrCylAction:=ADR(T_Station.THardware.TCylToolTension);
					iSelectedCylinder:=1;
					IF (T_Visu.T_PlcParam.dwActualPage = 230) THEN
						IF (T_Visu.ptrT_ExchgParam^.T_Cylinder.iSelectCylinder_Sonder1 = 1) THEN
							ptrCylAction:=ADR(T_Station.THardware.TCylToolTension);
							iSelectedCylinder:=1;
						ELSIF (T_Visu.ptrT_ExchgParam^.T_Cylinder.iSelectCylinder_Sonder1 = 2) THEN
							ptrCylAction:=ADR(T_Station.THardware.TCylToolLeftActive);
							iSelectedCylinder:=2;
						ELSIF (T_Visu.ptrT_ExchgParam^.T_Cylinder.iSelectCylinder_Sonder1 = 3) THEN
							ptrCylAction:=ADR(T_Station.THardware.TCylToolRightActive);
							iSelectedCylinder:=3;
						ELSIF (T_Visu.ptrT_ExchgParam^.T_Cylinder.iSelectCylinder_Sonder1 = 4) THEN
							ptrCylAction:=ADR(T_Station.THardware.TCylToolCenterActive);
							iSelectedCylinder:=4;
						ELSIF (T_Visu.ptrT_ExchgParam^.T_Cylinder.iSelectCylinder_Sonder1 = 5) THEN
							ptrCylAction:=ADR(T_Station.THardware.TCylToolPrismaLeftActive);
							iSelectedCylinder:=5;
						ELSIF (T_Visu.ptrT_ExchgParam^.T_Cylinder.iSelectCylinder_Sonder1 = 6) THEN
							ptrCylAction:=ADR(T_Station.THardware.TCylToolPrismaRightActive);
							iSelectedCylinder:=6;
						ELSE
							ptrCylAction:=ADR(T_Station.THardware.TCylToolTension);
							iSelectedCylinder:=1;
						END_IF;
					END_IF;
					(*Set pointer -->selection by the extern buttons*)
					IF (T_Visu.T_CtrleAction.iFunction = 510) THEN ptrCylAction:=ADR(T_Station.THardware.TCylToolTension);iSelectedCylinder:=1; END_IF;
					IF (T_Visu.T_CtrleAction.iFunction = 511) THEN ptrCylAction:=ADR(T_Station.THardware.TCylToolLeftActive);iSelectedCylinder:=2; END_IF;
					IF (T_Visu.T_CtrleAction.iFunction = 512) THEN ptrCylAction:=ADR(T_Station.THardware.TCylToolRightActive);iSelectedCylinder:=3; END_IF;
					IF (T_Visu.T_CtrleAction.iFunction = 513) THEN ptrCylAction:=ADR(T_Station.THardware.TCylToolCenterActive);iSelectedCylinder:=4; END_IF;
					IF (T_Visu.T_CtrleAction.iFunction = 514) THEN ptrCylAction:=ADR(T_Station.THardware.TCylToolPrismaLeftActive);iSelectedCylinder:=5; END_IF;
					IF (T_Visu.T_CtrleAction.iFunction = 515) THEN ptrCylAction:=ADR(T_Station.THardware.TCylToolPrismaRightActive);iSelectedCylinder:=6; END_IF;
					IF ((T_Visu.T_CtrleAction.iFunction >= 510) AND (T_Visu.T_CtrleAction.iFunction <= 515)) THEN
						T_Visu.T_CtrleAction.iFunction:=501;
					 END_IF;
					CASE T_Visu.T_CtrleAction.iFunction OF
					501:		xToggleCylinderState:=TRUE;
							IF ( iSelectedCylinder = 1) THEN
								IF (T_Visu.T_PlcParam.dwActualPage = 220) THEN
									ptrCylAction^.T_CtrleCyl.T_AnalogCylinder.rForceIn:=T_Visu.ptrT_ExchgParam^.T_InfoValueCommon.rToolTensionForce;
								ELSE
									IF (T_Visu.ptrT_ExchgParam^.T_Cylinder.iSelectToolTensionForce < 2) THEN
										(* Process work force *)
										ptrCylAction^.T_CtrleCyl.T_AnalogCylinder.rForceIn:=T_NovRam.T_Data.T_ProcessImageData.T_ProcessPara.rToolTensionProcess;
									END_IF;
									IF (T_Visu.ptrT_ExchgParam^.T_Cylinder.iSelectToolTensionForce > 1) THEN
										(* Setup (Cylinder Force) Force *)
										ptrCylAction^.T_CtrleCyl.T_AnalogCylinder.rForceIn:=T_NovRam.T_Data.T_Standard.T_Cyl_ToolTension.rForce;
									END_IF;
								END_IF;
							END_IF;
							tTimeOutAction:=T#2s;
					(* ToolTens force + *)
					502:		xToolTensForceAdd:=TRUE;
							tTimeOutAction:=T#2s;
					(* ToolTens force ++ *)
					503:		xToolTensForceAddMore:=TRUE;
							tTimeOutAction:=T#2s;
					(* ToolTens force - *)
					504:		xToolTensForceSub:=TRUE;
							tTimeOutAction:=T#2s;
					(* ToolTens force -- *)
					505:		xToolTensForceSubMore:=TRUE;
							tTimeOutAction:=T#2s;
					(* DO NOT USE FUNCTION 510,511,512,513,514,515 *)
					END_CASE;
			(* All process station *)
			601..699:	T_Process.iFunctNr:=T_Visu.T_CtrleAction.iFunction - 600;
					xActionProcStation:=TRUE;
					tTimeOutAction:=T#2s;
			(* All process machine *)
			701..799:	T_Process.iFunctNr:=T_Visu.T_CtrleAction.iFunction - 700;
					xActionProcMachine:=TRUE;
					(* Ref timeout 120s *)
					IF T_Visu.T_CtrleAction.iFunction = 710 THEN  tTimeOutAction:=T#120s; ELSE tTimeOutAction:=T#0.5s; END_IF
			(* Stop process *)
			800:		xStopProcess:=TRUE;
					tTimeOutAction:=T#30s;
			(* Stop cycle *)
			801:		xAction_StopCycle:=TRUE;
					tTimeOutAction:=T#30s;
			(* Copy profile to process value *)
			1001:	xAction_CopyProfileToProcess:=TRUE;
					tTimeOutAction:=T#10s;
			(* Load profile to process image *)
			1002:	xAction_LoadProfileToProcessImage:=TRUE;
					tTimeOutAction:=T#5s;
			(* Save profile to File *)
			1003:	xAction_SaveProfileToFile:=TRUE;
					tTimeOutAction:=T#5s;
			(* Delete Profile *)
			1004:	xActionDeleteProfile:=TRUE;
					tTimeOutAction:=T#5s;
			(* Save NovRAM with confirmation *)
			1005:	xAction_SaveNovRAM:=TRUE;
					tTimeOutAction:=T#6s;
			(* Save NovRAM without confirmation *)
			1006:	xAction_SaveNovRAMWithoutConfirm:=TRUE;
					tTimeOutAction:=T#10s;
			(* change page *)
			10001..10999:	xNavPanelChangePage:=TRUE;
						tTimeOutAction:=T#3s;
		END_CASE;
		(* Init. variable *)
		T_Visu.T_CtrleAction.xDone:=FALSE;
		T_Visu.T_CtrleAction.xNotReady:=FALSE;
		T_Visu.T_CtrleAction.xErr:=FALSE;
		T_Visu.T_CtrleAction.udiErrorID:=0;
		iStepAction:=1;
		iStepActionNovRam:=1;
		xStepActionDone:=FALSE;
		IF tTimeOutAction <> T#0s THEN TimerAction(IN:=FALSE); END_IF
		(* exit FB *)
		RETURN;
	END_IF;

(* Timer action *)
	IF tTimeOutAction <> T#0s THEN TimerAction(IN:=TRUE,PT:=tTimeOutAction); END_IF
	RisingEdgeTimeOut(CLK:=TimerAction.Q);
	IF RisingEdgeTimeOut.Q AND NOT(T_Visu.T_CtrleAction.xDone) AND NOT(T_Visu.T_CtrleAction.xErr) THEN
	(* Timeout action activ *)
		T_Visu.T_CtrleAction.xExecute:=FALSE;
		T_Visu.T_CtrleAction.xDone:=TRUE;
		T_Visu.T_CtrleAction.xNotReady:=FALSE;
		T_Visu.T_CtrleAction.xErr:=FALSE;
		T_Visu.T_CtrleAction.udiErrorID:=16#0;
		(* call confirmation message *)
		T_Visu.ptrT_ExchgParam^.T_Visu.T_Message.iState:=102;
(*			:=iFctReturnConfMessage(iNumAction:=-1);*)
		(* exit FB, do not continue the execution of action! *)
		RETURN;
	END_IF
(************************************************************************************************************************************************************************)
(***************                                          end  of the management for call a function of the visualisation interface                                           ********************)
(************************************************************************************************************************************************************************)

(************************************************************************************************************************************************************************)
(***************                                                   start of the checking of the activation of an visualisation action                                                   ********************)
(************************************************************************************************************************************************************************)
(* check if Action is Acitve and if the power supply is on, otherwise block the action *)
	xTmp:=	xStopAxis OR xMoveRelPosition OR xMoveAbsPosition OR xMoveContinousVel OR xSwitchMasterSlave OR xToggleAxisPower OR xResetAxis OR xReferenceAxis OR xTeachPosition;
	xTmp:=	xTmp OR xToggleCylinderState OR xToolTensForceAdd OR xToolTensForceAddMore OR xToolTensForceSub OR xToolTensForceSubMore;
	xTmp:=	xTmp OR xToolFeederMoveStartPos OR xToggleAllAxisPower OR xCalcAngleRefIndex OR xToolFeederMoveLoadPos;
	xTmp:=	xTmp OR xActivateStationFunction OR xActionProcStation OR xActionProcMachine OR xStopProcess;
	xTmp:=	xTmp OR xOverlayGrindFeedSetPlung OR xOverlayMeasureToolDia OR xFctCorrectionToolDiameter OR xAction_LoadProfileToProcessImage;
	xTmp:=	xTmp OR ((T_Visu.T_PlcParam.dwActualPage = 430) AND xAction_SaveNovRAM);
(*SOA 31.01.2023  { *)
	xTmp:= xTmp OR (T_Visu.T_PlcParam.dwActualPage = 141) ;
(*SOA 31.01.2023  } *)
	IF xTmp THEN
		IF NOT(T_TwinSafeOut.QxContactor_K3) OR NOT(T_TwinSafeOut.QxContactor_K4) THEN
			xStopAxis:=xMoveRelPosition:=xMoveAbsPosition:=xMoveContinousVel:=xSwitchMasterSlave:=xToggleAxisPower:=xResetAxis:=xReferenceAxis:=xTeachPosition:=FALSE;
			xToggleCylinderState:=xToolTensForceAdd:=xToolTensForceAddMore:=xToolTensForceSub:=xToolTensForceSubMore:=FALSE;
			xToolFeederMoveStartPos:=xToggleAllAxisPower:=xCalcAngleRefIndex:=xToolFeederMoveLoadPos:= FALSE;
			xActivateStationFunction:=xActionProcStation:=xActionProcMachine:=xStopProcess:=FALSE;
			xOverlayGrindFeedSetPlung:=xOverlayMeasureToolDia:=xFctCorrectionToolDiameter:=xAction_LoadProfileToProcessImage:=FALSE;
			T_Visu.ptrT_ExchgParam^.T_FunctionCommon.xOpenOverlayMessageBox:=FALSE;
			T_Visu.ptrT_ExchgParam^.T_FunctionCommon.xOpenOverlayMeasureInput:=FALSE;
			T_Visu.ptrT_ExchgParam^.T_FunctionCommon.xOpenOverlaySetGrindPlunge:=FALSE;
			T_Visu.ptrT_ExchgParam^.T_FunctionCommon.xSaveButton:=FALSE;
			T_Visu.ptrT_ExchgParam^.T_FunctionCommon.xExitButton:=FALSE;
			T_Visu.ptrT_ExchgParam^.T_FunctionCommon.xHideProgressbar:=FALSE;
			xAction_SaveNovRAM:=FALSE;
			T_Visu.T_CtrleAction.xDone:=TRUE;
			T_Visu.T_CtrleAction.xNotReady:=FALSE;
			T_Visu.T_CtrleAction.xErr:=FALSE;
			T_Visu.T_CtrleAction.udiErrorID:=0;
			tTimeOutAction:=T#0s;
			TimerAction(IN:=FALSE);
			(* Display Message --> Switch first the energy supply ON *)
			T_ExchgParam.T_Visu.T_Message.iState:=120;
			xBlockConfirmMessage:=TRUE;
			TONTimeWaitMsg(IN:=FALSE);
		END_IF;
	END_IF;
	IF (T_ExchgParam.T_Visu.T_Message.iState = 120) THEN
		TONTimeWaitMsg(IN:=TRUE,PT:=T#3s);
		IF TONTimeWaitMsg.Q THEN
			T_ExchgParam.T_Visu.T_Message.iState:=0;	(* Deactivate again the message *)
		END_IF;
	ELSE
		TONTimeWaitMsg(IN:=FALSE);
	END_IF;

(* check if an error is active, otherwise block the action *)
	IF (T_ExchgParam.T_Visu.T_Message.iState = 401) THEN
		xTmp:=	xStopAxis OR xMoveRelPosition OR xMoveAbsPosition OR xMoveContinousVel OR xSwitchMasterSlave OR xToggleAxisPower OR xResetAxis OR xReferenceAxis OR xTeachPosition;
		xTmp:=	xTmp OR xToggleCylinderState OR xToolTensForceAdd OR xToolTensForceAddMore OR xToolTensForceSub OR xToolTensForceSubMore;
		xTmp:=	xTmp OR xToolFeederMoveStartPos OR xToggleAllAxisPower OR xCalcAngleRefIndex OR xToolFeederMoveLoadPos;
		xTmp:=	xTmp OR xActivateStationFunction OR xActionProcStation OR xActionProcMachine OR xStopProcess;
		xTmp:=	xTmp OR xOverlayGrindFeedSetPlung OR xOverlayMeasureToolDia OR xFctCorrectionToolDiameter OR xAction_LoadProfileToProcessImage;
		xTmp:=	xTmp OR ((T_Visu.T_PlcParam.dwActualPage = 430) AND xAction_SaveNovRAM);
		IF xTmp THEN
			xStopAxis:=xMoveRelPosition:=xMoveAbsPosition:=xMoveContinousVel:=xSwitchMasterSlave:=xToggleAxisPower:=xResetAxis:=xReferenceAxis:=xTeachPosition:=FALSE;
			xToggleCylinderState:=xToolTensForceAdd:=xToolTensForceAddMore:=xToolTensForceSub:=xToolTensForceSubMore:=FALSE;
			xToolFeederMoveStartPos:=xToggleAllAxisPower:=xCalcAngleRefIndex:=xToolFeederMoveLoadPos:=FALSE;
			xActivateStationFunction:=xActionProcStation:=xActionProcMachine:=xStopProcess:=FALSE;
			xOverlayGrindFeedSetPlung:=xOverlayMeasureToolDia:=xFctCorrectionToolDiameter:=xAction_LoadProfileToProcessImage:=FALSE;
			xAction_SaveNovRAM:=FALSE;
			T_Visu.T_CtrleAction.xDone:=TRUE;
			T_Visu.T_CtrleAction.xNotReady:=FALSE;
			T_Visu.T_CtrleAction.xErr:=FALSE;
			T_Visu.T_CtrleAction.udiErrorID:=0;
			tTimeOutAction:=T#0s;
			TimerAction(IN:=FALSE);
		END_IF;
	END_IF;
(************************************************************************************************************************************************************************)
(***************                                                   end of the checking of the activation of an visualisation action                                                   ********************)
(************************************************************************************************************************************************************************)

(************************************************************************************************************************************************************************)
(***************                                             start for the section for defined function of the visualisation interface                                               ********************)
(************************************************************************************************************************************************************************)
(* Action set parameter page *)
	IF xSetParameterPage THEN
		(* set parameter page *)
		CASE iStepAction OF
		(* check visu *)
		1:	IF (T_Visu.T_PlcParam.dwActualPage = 140) OR (T_Visu.T_PlcParam.dwActualPage = 150) THEN
				(* For this page. for select the parameter list, it need the system level *)
				IF (T_ExchgParam.T_Visu.T_Level.iActLevel <> 2) THEN
					T_ExchgParam.T_Visu.T_Message.iState:=36;	(* Display Message --> This parameter can be change only with system level *)
						T_Visu.ptrT_ExchgParam^.T_TouchScreenBtPanel.iStateBtLeft:=WORD_TO_INT(INT_TO_WORD(T_Visu.ptrT_ExchgParam^.T_TouchScreenBtPanel.iStateBtLeft) AND 16#FFEF);
				END_IF;
			END_IF;
			IF (T_ExchgParam.T_Visu.T_Message.iState <> 36) THEN
				xTmp:=	T_Visu.T_CtrleVisu.xDone
						AND NOT(T_Visu.T_CtrleVisu.xExecute)
						AND NOT(T_Visu.T_CtrleVisu.xErr);
				IF xTmp THEN
					(* next Step *)
					iStepAction :=10;
					xStepActionDone:=FALSE;
				(* activ error *)
				ELSE iStepAction:=95; END_IF
			ELSE
				iStepAction:=90;
			END_IF;
		(* Set parameter page *)
		10:	T_Visu.ptrT_ExchgParam^.T_Config.xBlockParaListNavi:=FALSE;
			T_Visu.ptrT_ExchgParam^.T_Config.xBlockParaListNavi1:=TRUE;
			T_Visu.ptrT_ExchgParam^.T_Config.xBlockProfilList:=TRUE;
			CASE T_Visu.ptrT_ExchgParam^.T_Visu.bActivSpecialLayer OF
				1:	T_Visu.T_PlcParam.dwSetNewPage:=170;
					T_Visu.ptrT_ExchgParam^.T_Config.iEditParam:=iFctGetEditParaList(	dwActualPage:=wSpecialLayerGeneralActivPage,
																				xMicroRodActive:=xMicroRodActive,
																				iSelectParaList:=T_Visu.ptrT_ExchgParam^.T_Config.iSelectParaList,
																				iSelectParaListTeachRot:=T_Visu.ptrT_ExchgParam^.T_Config.iSelectParaListTeachRot);
					IF (T_Visu.ptrT_ExchgParam^.T_Config.iEditParam = 140) OR (T_Visu.ptrT_ExchgParam^.T_Config.iEditParam = 150) THEN
						(* For this page. for select the parameter list, it need the system level *)
						IF (T_ExchgParam.T_Visu.T_Level.iActLevel <> 2) THEN
							T_ExchgParam.T_Visu.T_Message.iState:=36;	(* Display Message --> This parameter can be change only with system level *)
								T_Visu.ptrT_ExchgParam^.T_TouchScreenBtPanel.iStateBtLeft:=WORD_TO_INT(INT_TO_WORD(T_Visu.ptrT_ExchgParam^.T_TouchScreenBtPanel.iStateBtLeft) AND 16#FFEF);
								T_Visu.T_PlcParam.dwSetNewPage:=wSpecialLayerGeneralActivPage;
						END_IF;
					END_IF;
					IF (T_ExchgParam.T_Visu.T_Message.iState <> 36) THEN
						(* 09.12.2010 KFS:	{	*)
						IF (T_ExchgParam.T_Visu.T_Level.iActLevel =2) THEN
						(* 09.12.2010 KFS:	}	*)
							IF (T_Visu.ptrT_ExchgParam^.T_Config.iEditParam = 110) OR (T_Visu.ptrT_ExchgParam^.T_Config.iEditParam = 111) THEN
								T_Visu.ptrT_ExchgParam^.T_Config.xBlockProfilList:=FALSE;
							END_IF;
							IF ((T_Visu.ptrT_ExchgParam^.T_Config.iEditParam >= 120) AND (T_Visu.ptrT_ExchgParam^.T_Config.iEditParam <= 129)) THEN
								T_Visu.ptrT_ExchgParam^.T_Config.xBlockProfilList:=FALSE;
							END_IF;
							IF (T_Visu.ptrT_ExchgParam^.T_Config.iEditParam = 130) OR (T_Visu.ptrT_ExchgParam^.T_Config.iEditParam = 131) THEN
								T_Visu.ptrT_ExchgParam^.T_Config.xBlockParaListNavi1:=FALSE;
								T_Visu.ptrT_ExchgParam^.T_Config.xBlockParaListNavi:=TRUE;
								T_Visu.ptrT_ExchgParam^.T_Config.xBlockProfilList:=FALSE;
								(*  Set Loaded Profil Data from the read file*)
								T_Visu.ptrT_ExchgParam^.T_StationCommon.T_AutoGeometryPara:=T_NovRAM.T_Data.T_ProcessImageLoadData.T_AutoGeometryPara;
								T_Visu.ptrT_ExchgParam^.T_StationCommon.T_AutoGroovePara:=T_NovRAM.T_Data.T_ProcessImageLoadData.T_AutoGroovePara;
								T_Visu.ptrT_ExchgParam^.T_StationCommon.T_CalibrationPara:=T_NovRAM.T_Data.T_ProcessImageLoadData.T_CalibrationPara;
								T_Visu.ptrT_ExchgParam^.T_StationCommon.T_ProcessPara:=T_NovRAM.T_Data.T_ProcessImageLoadData.T_ProcessPara;
								T_Visu.ptrT_ExchgParam^.T_GeometryCommon.T_Geometry:=T_NovRAM.T_Data.T_ProcessImageLoadData.T_GeometryPara;
								T_Visu.ptrT_ExchgParam^.T_StationCommon.T_PrismPara:=T_NovRAM.T_Data.T_ProcessImageLoadData.T_PrismPara;
							END_IF;
							IF (T_Visu.ptrT_ExchgParam^.T_Config.iEditParam = 150) THEN
								T_Visu.ptrT_ExchgParam^.T_Config.xBlockParaListNavi:=TRUE;
							END_IF;
						(* 09.12.2010 KFS:	{	*)
						ELSE
							IF (T_Visu.ptrT_ExchgParam^.T_Config.iEditParam = 110) OR (T_Visu.ptrT_ExchgParam^.T_Config.iEditParam = 111) THEN
								IF  (T_Visu.ptrT_ExchgParam^.T_Config.iEditParam = 111) THEN
									 T_Visu.ptrT_ExchgParam^.T_Config.iEditParam:= 112;
								END_IF;
								T_Visu.ptrT_ExchgParam^.T_Config.xBlockProfilList:=FALSE;
							END_IF;
							IF ((T_Visu.ptrT_ExchgParam^.T_Config.iEditParam >= 120) AND (T_Visu.ptrT_ExchgParam^.T_Config.iEditParam <= 129)) THEN
								IF  (T_Visu.ptrT_ExchgParam^.T_Config.iEditParam = 121) THEN
									 T_Visu.ptrT_ExchgParam^.T_Config.iEditParam:= 126;
								ELSIF ( T_Visu.ptrT_ExchgParam^.T_Config.iEditParam = 123) THEN
									 T_Visu.ptrT_ExchgParam^.T_Config.iEditParam:= 127;
								ELSIF ( T_Visu.ptrT_ExchgParam^.T_Config.iEditParam = 125) THEN
									 T_Visu.ptrT_ExchgParam^.T_Config.iEditParam:= 128;
								END_IF;
								T_Visu.ptrT_ExchgParam^.T_Config.xBlockProfilList:=FALSE;
							END_IF;
							IF (T_Visu.ptrT_ExchgParam^.T_Config.iEditParam = 130) OR (T_Visu.ptrT_ExchgParam^.T_Config.iEditParam = 131) THEN
								T_Visu.ptrT_ExchgParam^.T_Config.xBlockParaListNavi1:=FALSE;
								T_Visu.ptrT_ExchgParam^.T_Config.xBlockParaListNavi:=TRUE;
								T_Visu.ptrT_ExchgParam^.T_Config.xBlockProfilList:=FALSE;
								(*  Set Loaded Profil Data from the read file*)
								T_Visu.ptrT_ExchgParam^.T_StationCommon.T_AutoGeometryPara:=T_NovRAM.T_Data.T_ProcessImageLoadData.T_AutoGeometryPara;
								T_Visu.ptrT_ExchgParam^.T_StationCommon.T_AutoGroovePara:=T_NovRAM.T_Data.T_ProcessImageLoadData.T_AutoGroovePara;
								T_Visu.ptrT_ExchgParam^.T_StationCommon.T_CalibrationPara:=T_NovRAM.T_Data.T_ProcessImageLoadData.T_CalibrationPara;
								T_Visu.ptrT_ExchgParam^.T_StationCommon.T_ProcessPara:=T_NovRAM.T_Data.T_ProcessImageLoadData.T_ProcessPara;
								T_Visu.ptrT_ExchgParam^.T_GeometryCommon.T_Geometry:=T_NovRAM.T_Data.T_ProcessImageLoadData.T_GeometryPara;
								T_Visu.ptrT_ExchgParam^.T_StationCommon.T_PrismPara:=T_NovRAM.T_Data.T_ProcessImageLoadData.T_PrismPara;
							END_IF;
							IF (T_Visu.ptrT_ExchgParam^.T_Config.iEditParam = 150) THEN
								T_Visu.ptrT_ExchgParam^.T_Config.xBlockParaListNavi:=TRUE;
							END_IF;
						END_IF;
						(* 09.12.2010 KFS:	}	*)
					END_IF;
				2:	T_Visu.T_PlcParam.dwSetNewPage:=270;
					T_Visu.ptrT_ExchgParam^.T_Config.iEditParam:=iFctGetEditParaList(	dwActualPage:=wSpecialLayerToolRotActivPage,
																				xMicroRodActive:=xMicroRodActive,
																				iSelectParaList:=T_Visu.ptrT_ExchgParam^.T_Config.iSelectParaList,
																				iSelectParaListTeachRot:=T_Visu.ptrT_ExchgParam^.T_Config.iSelectParaListTeachRot);
				3:	T_Visu.T_PlcParam.dwSetNewPage:=370;
					T_Visu.ptrT_ExchgParam^.T_Config.iEditParam:=iFctGetEditParaList(	dwActualPage:=wSpecialLayerWireFeedActivPage,
																				xMicroRodActive:=xMicroRodActive,
																				iSelectParaList:=T_Visu.ptrT_ExchgParam^.T_Config.iSelectParaList,
																				iSelectParaListTeachRot:=T_Visu.ptrT_ExchgParam^.T_Config.iSelectParaListTeachRot);
				4:	T_Visu.T_PlcParam.dwSetNewPage:=470;
					T_Visu.ptrT_ExchgParam^.T_Config.iEditParam:=iFctGetEditParaList(	dwActualPage:=wSpecialLayerGrindAxisActivPage,
																				xMicroRodActive:=xMicroRodActive,
																				iSelectParaList:=T_Visu.ptrT_ExchgParam^.T_Config.iSelectParaList,
																				iSelectParaListTeachRot:=T_Visu.ptrT_ExchgParam^.T_Config.iSelectParaListTeachRot);
			END_CASE;
			T_Visu.T_CtrleVisu.iFunction:=1;
			T_Visu.T_CtrleVisu.xExecute:=TRUE;
			(* activ step *)
			iStepAction:=20;
			xStepActionDone:=FALSE;
		(* wait for changing page *)
		20:	IF NOT(xStepActionDone) THEN
			(* release execution *)
				T_Visu.T_CtrleVisu.xExecute:=FALSE;
				(* confirm step done *)
				xStepActionDone:=TRUE;
			ELSE
				IF T_Visu.T_CtrleVisu.xDone THEN
				(* activ next step *)
					iStepAction:=90;
					xStepActionDone:=FALSE;
				END_IF
				IF T_Visu.T_CtrleVisu.xErr THEN
				(* activ next error *)
					iStepAction:=99;
					xStepActionDone:=FALSE;
				END_IF
			END_IF
		(* change page done *)
		90:	T_Visu.T_CtrleAction.xDone:=TRUE;
			T_Visu.T_CtrleAction.xNotReady:=FALSE;
			T_Visu.T_CtrleAction.xErr:=FALSE;
			T_Visu.T_CtrleAction.udiErrorID:=0;
			xSetParameterPage:=FALSE;
		(* override done *)
		91:	T_Visu.T_CtrleAction.xDone:=TRUE;
			T_Visu.T_CtrleAction.xNotReady:=FALSE;
			T_Visu.T_CtrleAction.xErr:=FALSE;
			T_Visu.T_CtrleAction.udiErrorID:=0;
			xSetParameterPage:=FALSE;
		(* not ready *)
		95:	T_Visu.T_CtrleAction.xDone:=TRUE;
			T_Visu.T_CtrleAction.xNotReady:=FALSE;
			T_Visu.T_CtrleAction.xErr:=FALSE;
			T_Visu.T_CtrleAction.udiErrorID:=0;
			xSetParameterPage:=FALSE;
		(* error *)
		99:	T_Visu.T_CtrleAction.xDone:=FALSE;
			T_Visu.T_CtrleAction.xNotReady:=FALSE;
			T_Visu.T_CtrleAction.xErr:=TRUE;
			T_Visu.T_CtrleAction.udiErrorID:=16#F0000 + T_Visu.T_CtrleAction.iFunction;
			xSetParameterPage:=FALSE;
		END_CASE
	END_IF

(* Action change page from navigation panel *)
	IF xNavPanelChangePage OR xBtPanelLeftChangePage OR  xBtPanelRightChangePage OR xNextPageVertical THEN
		(* Step change page from navigation panel *)
		CASE iStepAction OF
		(* check visu *)
		1:	xTmp:=	T_Visu.T_CtrleVisu.xDone
					AND NOT(T_Visu.T_CtrleVisu.xExecute)
					AND NOT(T_Visu.T_CtrleVisu.xErr);
			IF xTmp THEN
				(* next Step *)
				iStepAction :=10;
				xStepActionDone:=FALSE;
			(* activ error *)
			ELSE iStepAction:=95; END_IF
		(* activ change page *)
		10:	T_Visu.T_CtrleVisu.xExecute:=TRUE;
			T_Visu.T_CtrleVisu.iFunction:=1;
			T_Visu.ptrT_ExchgParam^.T_Config.iEditParam:=0;
			IF xNavPanelChangePage THEN
				T_Visu.T_PlcParam.dwSetNewPage:=INT_TO_DWORD(T_Visu.T_CtrleAction.iFunction - 10000);
				CASE T_Visu.ptrT_ExchgParam^.T_Visu.bActivSpecialLayer OF
					0:	IF awNormalLayerActivPage[wTmpNormalLayerActivTask] <> 0 AND awNormalLayerActivPage[wTmpNormalLayerActivTask] <> T_Visu.T_PlcParam.dwSetNewPage THEN
							T_Visu.T_PlcParam.dwSetNewPage:=awNormalLayerActivPage[wTmpNormalLayerActivTask];
						END_IF;
					1:	IF awSpecialLayerGeneralActivPage[wTmpSpecialLayerGeneralActivTask] <> 0 AND awSpecialLayerGeneralActivPage[wTmpSpecialLayerGeneralActivTask] <> T_Visu.T_PlcParam.dwSetNewPage THEN
							T_Visu.T_PlcParam.dwSetNewPage:=awSpecialLayerGeneralActivPage[wTmpSpecialLayerGeneralActivTask];
						END_IF;
					2:	IF awSpecialLayerToolRotActivPage[wTmpSpecialLayerToolRotActivTask] <> 0 AND awSpecialLayerToolRotActivPage[wTmpSpecialLayerToolRotActivTask] <> T_Visu.T_PlcParam.dwSetNewPage THEN
							T_Visu.T_PlcParam.dwSetNewPage:=awSpecialLayerToolRotActivPage[wTmpSpecialLayerToolRotActivTask];
						END_IF;
					3:	IF awSpecialLayerWireFeedActivPage[wTmpSpecialLayerWireFeedActivTask] <> 0 AND awSpecialLayerWireFeedActivPage[wTmpSpecialLayerWireFeedActivTask] <> T_Visu.T_PlcParam.dwSetNewPage THEN
							T_Visu.T_PlcParam.dwSetNewPage:=awSpecialLayerWireFeedActivPage[wTmpSpecialLayerWireFeedActivTask];
						END_IF;
					4:	IF awSpecialLayerGrindAxisActivPage[wTmpSpecialLayerGrindAxisActivTask] <> 0 AND awSpecialLayerGrindAxisActivPage[wTmpSpecialLayerGrindAxisActivTask] <> T_Visu.T_PlcParam.dwSetNewPage THEN
							T_Visu.T_PlcParam.dwSetNewPage:=awSpecialLayerGrindAxisActivPage[wTmpSpecialLayerGrindAxisActivTask];
						END_IF;
				END_CASE;
			END_IF;
			IF xBtPanelLeftChangePage THEN
				T_Visu.T_PlcParam.dwSetNewPage:=dwSetNewPage;
				T_Visu.ptrT_ExchgParam^.T_Config.xBlockParaListNavi:=FALSE;
				T_Visu.ptrT_ExchgParam^.T_Config.xBlockParaListNavi1:=TRUE;
				T_Visu.ptrT_ExchgParam^.T_Config.xBlockProfilList:=TRUE;
			END_IF;
(*SOA*)
			IF xBtPanelRightChangePage THEN
				T_Visu.T_PlcParam.dwSetNewPage:=dwSetNewPage;
				T_Visu.ptrT_ExchgParam^.T_Config.xBlockParaListNavi:=FALSE;
				T_Visu.ptrT_ExchgParam^.T_Config.xBlockParaListNavi1:=TRUE;
				T_Visu.ptrT_ExchgParam^.T_Config.xBlockProfilList:=TRUE;
			END_IF;
(*SOA*)
			IF xNextPageVertical THEN
				IF (T_Visu.T_PageIndex[T_Visu.T_PlcParam.dwActualPage + 1].iIndexConfigPage <> 0) THEN
					T_Visu.T_PlcParam.dwSetNewPage:=T_Visu.T_PlcParam.dwActualPage + 1;
				ELSE
					FOR ii:=1 TO 9 DO
						IF (T_Visu.T_PageIndex[T_Visu.T_PlcParam.dwActualPage - 1].iIndexConfigPage <> 0) THEN
							T_Visu.T_PlcParam.dwActualPage:=T_Visu.T_PlcParam.dwActualPage - 1;
						ELSE
							T_Visu.T_PlcParam.dwSetNewPage:=T_Visu.T_PlcParam.dwActualPage;
							EXIT;
						END_IF;
					END_FOR;
				END_IF;
				CASE T_Visu.ptrT_ExchgParam^.T_Visu.bActivSpecialLayer OF
					0:	awNormalLayerActivPage[wTmpNormalLayerActivTask]:=DWORD_TO_WORD(T_Visu.T_PlcParam.dwSetNewPage);
					1:	awSpecialLayerGeneralActivPage[wTmpSpecialLayerGeneralActivTask]:=DWORD_TO_WORD(T_Visu.T_PlcParam.dwSetNewPage);
					2:	awSpecialLayerToolRotActivPage[wTmpSpecialLayerToolRotActivTask]:=DWORD_TO_WORD(T_Visu.T_PlcParam.dwSetNewPage);
					3:	awSpecialLayerWireFeedActivPage[wTmpSpecialLayerWireFeedActivTask]:=DWORD_TO_WORD(T_Visu.T_PlcParam.dwSetNewPage);
					4:	awSpecialLayerGrindAxisActivPage[wTmpSpecialLayerGrindAxisActivTask]:=DWORD_TO_WORD(T_Visu.T_PlcParam.dwSetNewPage);
				END_CASE;
			END_IF;
			(* next Step *)
			iStepAction :=20;
			xStepActionDone:=FALSE;
		(* wait  confirmation *)
		20:	IF NOT(xStepActionDone) THEN
				T_Visu.T_CtrleVisu.xExecute:=FALSE;
				(* confirm Step *)
				xStepActionDone:=TRUE;
			ELSE
				IF T_Visu.T_CtrleVisu.xDone THEN
				(* next Step *)
					iStepAction :=90;
					xStepActionDone:=FALSE;
				ELSE	IF T_Visu.T_CtrleVisu.xErr THEN
							iStepAction:=99;
							xStepActionDone:=FALSE;
						END_IF
				END_IF
			END_IF
		(* change page done *)
		90:	T_Visu.T_CtrleAction.xDone:=TRUE;
			T_Visu.T_CtrleAction.xNotReady:=FALSE;
			T_Visu.T_CtrleAction.xErr:=FALSE;
			T_Visu.T_CtrleAction.udiErrorID:=0;
			xNavPanelChangePage:=FALSE;
			xBtPanelLeftChangePage:=FALSE;
			xBtPanelRightChangePage:=FALSE;
			xNextPageVertical:=FALSE;
		(* visu not ready *)
		95:	T_Visu.T_CtrleAction.xDone:=TRUE;
			T_Visu.T_CtrleAction.xNotReady:=FALSE;
			T_Visu.T_CtrleAction.xErr:=FALSE;
			T_Visu.T_CtrleAction.udiErrorID:=0;
			xNavPanelChangePage:=FALSE;
			xBtPanelLeftChangePage:=FALSE;
			xBtPanelRightChangePage:=FALSE;
			xNextPageVertical:=FALSE;
		(* error *)
		99:	T_Visu.T_CtrleAction.xDone:=FALSE;
			T_Visu.T_CtrleAction.xNotReady:=FALSE;
			T_Visu.T_CtrleAction.xErr:=TRUE;
			T_Visu.T_CtrleAction.udiErrorID:=16#F0000 + T_Visu.T_CtrleAction.iFunction;
			xNavPanelChangePage:=FALSE;
			xBtPanelLeftChangePage:=FALSE;
			xBtPanelRightChangePage:=FALSE;
			xNextPageVertical:=FALSE;
		END_CASE
	END_IF

(* Action reset error station *)
	IF xResetError THEN
		(* FB clear error station *)
		fbQvisClearError(	xExecute:=xResetError,
						iError:=T_Visu.T_CtrleAction.iFunction,
						T_Message:=T_ExchgParam.T_Visu.T_Message,
						T_Station:=T_Station,
						T_Process:=T_Process,
						T_NovRAM:=T_NovRAM,
						T_Profile:=T_Profile,
						T_HDD:=T_HDD,
						xDone=>T_Visu.T_CtrleAction.xDone,
						xNotReady=>T_Visu.T_CtrleAction.xNotReady,
						xErr=>T_Visu.T_CtrleAction.xErr,
						udiErrorID=>T_Visu.T_CtrleAction.udiErrorID);
		IF T_Visu.T_CtrleAction.xDone OR T_Visu.T_CtrleAction.xNotReady OR T_Visu.T_CtrleAction.xErr THEN
			xResetError:=FALSE;
			fbQvisClearError(	xExecute:=xResetError,
							iError:=T_Visu.T_CtrleAction.iFunction,
							T_Message:=T_ExchgParam.T_Visu.T_Message,
							T_Station:=T_Station,
							T_Process:=T_Process,
							T_NovRAM:=T_NovRAM,
							T_Profile:=T_Profile,
							T_HDD:=T_HDD);
		END_IF
	END_IF

(* Action Delete Errorlist for Machine and Station *)
	IF xDeleteErrorList THEN
		(* Step saving NovRAM *)
		CASE iStepAction OF
		(* check NovRAM *)
		1:	xTmp:=	T_NovRAM.T_Ctrle.xDone
					AND NOT(T_NovRAM.T_Ctrle.xExecute)
					AND NOT(T_NovRAM.T_Ctrle.xErr);
			IF xTmp THEN
				(* next Step *)
				iStepAction :=10;
			(* activ error *)
			ELSE iStepAction:=95; END_IF
		10:	(* For delete the error, it need the system level *)
			IF (T_ExchgParam.T_Visu.T_Level.iActLevel <> 2) THEN
				T_ExchgParam.T_Visu.T_Message.iState:=42;	(* Display Message --> The error list may delete only in system level ! *)
				iStepAction:=90;
				RETURN;
			END_IF;
			T_Visu.ptrT_ExchgParam^.T_Visu.T_Message.iState:=108;	(* Confirm saving action <Enter>, or escape <Esc> ? *)
			(* next Step *)
			iStepAction :=20;
		(* waiting for saving confirmation key <Enter> or <Esc> *)
		20:	IF RisingEdgeKeyPanel_Enter.Q THEN
			(* Display message *)
				T_Visu.ptrT_ExchgParam^.T_Visu.T_Message.iState:=13;	(* Start saving *)
				(* next step *)
				iStepAction:=30;
			ELSE
				IF RisingEdgeKeyPanel_Esc.Q THEN iStepAction:=90; END_IF
				(* An other message has been displayed, stop saving action *)
				IF T_Visu.ptrT_ExchgParam^.T_Visu.T_Message.iState<>108 THEN iStepAction:=90; END_IF
			END_IF
		30:	FOR ii:=1 TO 20 DO
				T_NovRAM.T_Data.T_ErrorNrList.adiErrorListMachine[ii]:=0;
				T_NovRAM.T_Data.T_ErrorNrList.asErrorTimeStampMachine[ii]:='';
			END_FOR;
			(* activ save *)
			T_NovRAM.T_Ctrle.xExecute:=TRUE;
			T_NovRAM.T_Ctrle.iFunction:=2;
			(* next Step *)
			iStepAction :=40;
			xStepActionDone:=FALSE;
		(* wait save confirmation *)
		40:	IF NOT(xStepActionDone) THEN
				T_NovRAM.T_Ctrle.xExecute:=FALSE;
				(* confirm Step *)
				xStepActionDone:=TRUE;
			ELSE
				IF T_NovRAM.T_Ctrle.xDone THEN
				(* next Step *)
					iStepAction :=90;
					xStepActionDone:=FALSE;
					xUpdateErrorList:=TRUE;
				ELSE	IF T_NovRAM.T_Ctrle.xErr THEN
							iStepAction:=99;
							xStepActionDone:=FALSE;
						END_IF
				END_IF
			END_IF
		(* no code, waiting timeout *)
		89:	IF TimerAction.Q THEN iStepAction:=90; END_IF
		(* save done *)
		90:	IF (T_ExchgParam.T_Visu.T_Message.iState <> 42) THEN
				T_Visu.ptrT_ExchgParam^.T_Visu.T_Message.iState:=0;
			END_IF;
			T_Visu.T_CtrleAction.xDone:=TRUE;
			T_Visu.T_CtrleAction.xNotReady:=FALSE;
			T_Visu.T_CtrleAction.xErr:=FALSE;
			T_Visu.T_CtrleAction.udiErrorID:=0;
			xDeleteErrorList:=FALSE;
		(* NovRAM not ready *)
		95:	TimerNotReady(IN:=TRUE);
			xDeleteErrorList:=FALSE;
		(* error *)
		99:	T_Visu.T_CtrleAction.xDone:=FALSE;
			T_Visu.T_CtrleAction.xNotReady:=FALSE;
			T_Visu.T_CtrleAction.xErr:=TRUE;
			T_Visu.T_CtrleAction.udiErrorID:=16#F0000 + T_Visu.T_CtrleAction.iFunction;
			xDeleteErrorList:=FALSE;
		END_CASE;
	END_IF;

(* Open Overlay for input measured tool diameter *)
	IF xOverlayMeasureToolDia THEN
		CASE iStepAction OF
		(* check axis *)
		1:	IF NOT T_Station.TControl.xHardwareConfigError THEN
				xStepActionDone:=FALSE;
				iStepAction:=95;
				xTmp:=	T_Station.THardware.TAxisGrindFeeder.T_CtrleSingle.xDone
						AND T_Station.THardware.TAxisGrindFeeder.T_CtrleSingle.xReady
						AND T_Station.THardware.TAxisGrindFeeder.T_CtrleSingle.xNotMoving
						AND NOT(T_Station.THardware.TAxisGrindFeeder.T_CtrleSingle.xErr)
						AND NOT(T_Station.THardware.TAxisGrindFeeder.T_CtrleSingle.xExecute);
				(* Start/Stop position or speed of teachin page has to be confirmed *)
				IF xTmp THEN
					iStepAction:=10;
				END_IF
			ELSE
				iStepAction:=95;
			END_IF;
		10:	(* Open Overlay *)
			T_Visu.ptrT_ExchgParam^.T_FunctionCommon.xOpenOverlayMeasureInput:=TRUE;
			T_Visu.ptrT_ExchgParam^.T_FunctionCommon.xHideProgressbar:=TRUE;
			T_Visu.ptrT_ExchgParam^.T_FunctionCommon.rInputMeasToolDiameter:=T_Visu.ptrT_ExchgParam^.T_InfoValueCommon.rToolDiameter;
			(* next Step *)
			iStepAction :=20;
		20:	IF T_Visu.ptrT_ExchgParam^.T_FunctionCommon.xSaveButton THEN
				T_Visu.ptrT_ExchgParam^.T_FunctionCommon.xSaveButton:=FALSE;
				T_Visu.ptrT_ExchgParam^.T_FunctionCommon.xExitButton:=FALSE;
				(* next Step *)
				iStepAction :=30;
			END_IF;
			IF T_Visu.ptrT_ExchgParam^.T_FunctionCommon.xExitButton THEN
				T_Visu.ptrT_ExchgParam^.T_FunctionCommon.xSaveButton:=FALSE;
				T_Visu.ptrT_ExchgParam^.T_FunctionCommon.xExitButton:=FALSE;
				(* next Step *)
				iStepAction :=90;
			END_IF;
			IF T_Visu.T_CtrleAction.xDone THEN
				T_Visu.ptrT_ExchgParam^.T_FunctionCommon.xOpenOverlayMeasureInput:=FALSE;
				T_Visu.ptrT_ExchgParam^.T_FunctionCommon.xSaveButton:=FALSE;
				T_Visu.ptrT_ExchgParam^.T_FunctionCommon.xExitButton:=FALSE;
				T_Visu.ptrT_ExchgParam^.T_FunctionCommon.xHideProgressbar:=FALSE;
				xOverlayMeasureToolDia:=FALSE;
			END_IF;
		(* activ function axis *)
		30:	T_Station.THardware.TAxisGrindFeeder.T_CtrleSingle.rSetPosition:=	T_Station.THardware.TAxisGrindFeeder.T_LiveValue.lrActualPosition +
																		(T_Visu.ptrT_ExchgParam^.T_FunctionCommon.rInputMeasToolDiameter -
																		T_Visu.ptrT_ExchgParam^.T_InfoValueCommon.rToolDiameter);
			IF (T_Station.THardware.TAxisGrindFeeder.T_CtrleSingle.rSetPosition < T_NovRAM.T_Data.T_ProcessImageData.T_PrismPara.rToolDiameterMin) OR
			     (T_Station.THardware.TAxisGrindFeeder.T_CtrleSingle.rSetPosition > (T_NovRAM.T_Data.T_ProcessImageData.T_PrismPara.rToolDiameterMax + T_NovRAM.T_Data.T_Standard.T_TeachINGrindFeeder.rOffsetSWPosEndSwitch)) THEN
				T_Visu.ptrT_ExchgParam^.T_Visu.T_Message.iState:=123;	(* Out of Range, GrindFeeder position not settled! *)
				iStepAction:=50;
			ELSE
				T_Station.THardware.TAxisGrindFeeder.T_CtrleSingle.iFunction:=11;
				T_Station.THardware.TAxisGrindFeeder.T_CtrleSingle.xExecute:=TRUE;
				(* next step *)
				iStepAction:=50;
			END_IF;
			xStepActionDone:=FALSE;
		(* confirm execution *)
		50:	IF NOT(xStepActionDone) THEN
			(* confirm execution *)
				T_Station.THardware.TAxisGrindFeeder.T_CtrleSingle.xExecute:=FALSE;
				xStepActionDone:=TRUE;
			ELSE
				IF T_Station.THardware.TAxisGrindFeeder.T_CtrleSingle.xDone THEN
				(* confirm action next step *)
					iStepAction:=90;
					xStepActionDone:=FALSE;
				ELSE
					IF T_Station.THardware.TAxisGrindFeeder.T_CtrleSingle.xErr THEN
					(* activ action not ready or error *)
						iStepAction:=99;
						xStepActionDone:=FALSE;
					END_IF
				END_IF
			END_IF
		(* action done *)
		90:	T_Visu.ptrT_ExchgParam^.T_StationCommon.wState:=T_Visu.ptrT_ExchgParam^.T_StationCommon.wState AND 16#BF;
			T_Visu.T_CtrleAction.xDone:=TRUE;
			T_Visu.T_CtrleAction.xNotReady:=FALSE;
			T_Visu.T_CtrleAction.xErr:=FALSE;
			T_Visu.T_CtrleAction.udiErrorID:=0;
			xOverlayMeasureToolDia:=FALSE;
			T_Visu.ptrT_ExchgParam^.T_FunctionCommon.xOpenOverlayMeasureInput:=FALSE;
			T_Visu.ptrT_ExchgParam^.T_FunctionCommon.xHideProgressbar:=FALSE;
		(* axis not ready *)
		95:	T_Visu.ptrT_ExchgParam^.T_StationCommon.wState:=T_Visu.ptrT_ExchgParam^.T_StationCommon.wState AND 16#BF;
			TimerNotReady(IN:=TRUE);
			xOverlayMeasureToolDia:=FALSE;
			T_Visu.ptrT_ExchgParam^.T_FunctionCommon.xOpenOverlayMeasureInput:=FALSE;
			T_Visu.ptrT_ExchgParam^.T_FunctionCommon.xHideProgressbar:=FALSE;
		(* error *)
		99:	T_Visu.ptrT_ExchgParam^.T_StationCommon.wState:=T_Visu.ptrT_ExchgParam^.T_StationCommon.wState AND 16#BF;
			T_Visu.T_CtrleAction.xDone:=TRUE;
			T_Visu.T_CtrleAction.xNotReady:=FALSE;
			IF (T_Station.THardware.TAxisGrindFeeder.T_Config_Gen.iTyp <> 0) THEN
				diErrorNr:=(T_Station.THardware.TAxisGrindFeeder.T_Config_Gen.iTyp * 1000000) + T_Station.THardware.TAxisGrindFeeder.T_CtrleSingle.udiErrorID;
			ELSE
				diErrorNr:=0;
			END_IF;
			FBErrorMessage(	diErrorNr:=diErrorNr,
							T_ErrorList:=T_ErrorList);
			T_Visu.ptrT_ExchgParam^.T_Visu.T_Message.sDynamicTextEnglish:=FBErrorMessage.sErrorTextEnglish;
			T_Visu.ptrT_ExchgParam^.T_Visu.T_Message.sDynamicTextDeutsch:=FBErrorMessage.sErrorTextDeutsch;
			T_Visu.ptrT_ExchgParam^.T_Visu.T_Message.sDynamicTextFrancais:=FBErrorMessage.sErrorTextFrancais;
			T_Visu.ptrT_ExchgParam^.T_SafetyCtrl.xSetForceError:=TRUE;
			T_Visu.ptrT_ExchgParam^.T_SafetyCtrl.diSetForceErrorNr:=diErrorNr;
			T_Visu.T_CtrleAction.xErr:=FALSE;
			T_Visu.T_CtrleAction.udiErrorID:=0;
			T_Station.THardware.TAxisGrindFeeder.T_CtrleSingle.iFunction:=1;
			T_Station.THardware.TAxisGrindFeeder.T_CtrleSingle.xExecute:=TRUE;
			xOverlayMeasureToolDia:=FALSE;
			T_Visu.ptrT_ExchgParam^.T_FunctionCommon.xOpenOverlayMeasureInput:=FALSE;
			T_Visu.ptrT_ExchgParam^.T_FunctionCommon.xHideProgressbar:=FALSE;
		END_CASE
	END_IF;

(* Open Overlay for input the correction of the position of the GrindFeeder *)
	IF xOverlayGrindFeedSetPlung THEN
		CASE iStepAction OF
		(* check axis *)
		1:	IF NOT T_Station.TControl.xHardwareConfigError THEN
				xStepActionDone:=FALSE;
				iStepAction:=95;
				xTmp:=	T_Station.THardware.TAxisGrindFeeder.T_CtrleSingle.xDone
						AND T_Station.THardware.TAxisGrindFeeder.T_CtrleSingle.xReady
						AND T_Station.THardware.TAxisGrindFeeder.T_CtrleSingle.xNotMoving
						AND NOT(T_Station.THardware.TAxisGrindFeeder.T_CtrleSingle.xErr)
						AND NOT(T_Station.THardware.TAxisGrindFeeder.T_CtrleSingle.xExecute);
				(* Start/Stop position or speed of teachin page has to be confirmed *)
				IF xTmp THEN
					iStepAction:=10;
				END_IF
			ELSE
				iStepAction:=95;
			END_IF;
		10:	(* Open Overlay *)
			T_Visu.ptrT_ExchgParam^.T_FunctionCommon.xOpenOverlaySetGrindPlunge:=TRUE;
			T_Visu.ptrT_ExchgParam^.T_FunctionCommon.xHideProgressbar:=TRUE;
			T_Visu.ptrT_ExchgParam^.T_FunctionCommon.rInputGrindPlunge:=T_NovRAM.T_Data.T_ProcessImageData.T_CalibrationPara.rPlungeLengthGrindFeedCalib;
			(* next Step *)
			iStepAction :=20;
		20:	IF T_Visu.ptrT_ExchgParam^.T_FunctionCommon.xSaveButton THEN
				T_Visu.ptrT_ExchgParam^.T_FunctionCommon.xSaveButton:=FALSE;
				T_Visu.ptrT_ExchgParam^.T_FunctionCommon.xExitButton:=FALSE;
				(* next Step *)
				iStepAction :=30;
			END_IF;
			IF T_Visu.ptrT_ExchgParam^.T_FunctionCommon.xExitButton THEN
				T_Visu.ptrT_ExchgParam^.T_FunctionCommon.xSaveButton:=FALSE;
				T_Visu.ptrT_ExchgParam^.T_FunctionCommon.xExitButton:=FALSE;
				(* next Step *)
				iStepAction :=90;
			END_IF;
			IF T_Visu.T_CtrleAction.xDone THEN
				T_Visu.ptrT_ExchgParam^.T_FunctionCommon.xOpenOverlaySetGrindPlunge:=FALSE;
				T_Visu.ptrT_ExchgParam^.T_FunctionCommon.xSaveButton:=FALSE;
				T_Visu.ptrT_ExchgParam^.T_FunctionCommon.xExitButton:=FALSE;
				T_Visu.ptrT_ExchgParam^.T_FunctionCommon.xHideProgressbar:=FALSE;
				xOverlayGrindFeedSetPlung:=FALSE;
			END_IF;
		(* activ function axis *)
		30:	T_Station.THardware.TAxisGrindFeeder.T_CtrleSingle.rSetPosition:=	T_Station.THardware.TAxisGrindFeeder.T_LiveValue.lrActualPosition +
																		T_Visu.ptrT_ExchgParam^.T_FunctionCommon.rInputGrindPlunge;
			T_Station.THardware.TAxisGrindFeeder.T_CtrleSingle.iFunction:=11;
			T_Station.THardware.TAxisGrindFeeder.T_CtrleSingle.xExecute:=TRUE;
			(* next step *)
			iStepAction:=50;
			xStepActionDone:=FALSE;
		(* confirm execution *)
		50:	IF NOT(xStepActionDone) THEN
			(* confirm execution *)
				T_Station.THardware.TAxisGrindFeeder.T_CtrleSingle.xExecute:=FALSE;
				xStepActionDone:=TRUE;
			ELSE
				IF T_Station.THardware.TAxisGrindFeeder.T_CtrleSingle.xDone THEN
				(* confirm action next step *)
					iStepAction:=90;
					xStepActionDone:=FALSE;
				ELSE
					IF T_Station.THardware.TAxisGrindFeeder.T_CtrleSingle.xErr THEN
					(* activ action not ready or error *)
						iStepAction:=99;
						xStepActionDone:=FALSE;
					END_IF
				END_IF
			END_IF
		(* action done *)
		90:	T_Visu.ptrT_ExchgParam^.T_StationCommon.wState:=T_Visu.ptrT_ExchgParam^.T_StationCommon.wState AND 16#BF;
			T_Visu.T_CtrleAction.xDone:=TRUE;
			T_Visu.T_CtrleAction.xNotReady:=FALSE;
			T_Visu.T_CtrleAction.xErr:=FALSE;
			T_Visu.T_CtrleAction.udiErrorID:=0;
			xOverlayGrindFeedSetPlung:=FALSE;
			T_Visu.ptrT_ExchgParam^.T_FunctionCommon.xOpenOverlaySetGrindPlunge:=FALSE;
			T_Visu.ptrT_ExchgParam^.T_FunctionCommon.xHideProgressbar:=FALSE;
		(* axis not ready *)
		95:	T_Visu.ptrT_ExchgParam^.T_StationCommon.wState:=T_Visu.ptrT_ExchgParam^.T_StationCommon.wState AND 16#BF;
			TimerNotReady(IN:=TRUE);
			xOverlayGrindFeedSetPlung:=FALSE;
			T_Visu.ptrT_ExchgParam^.T_FunctionCommon.xOpenOverlaySetGrindPlunge:=FALSE;
			T_Visu.ptrT_ExchgParam^.T_FunctionCommon.xHideProgressbar:=FALSE;
		(* error *)
		99:	T_Visu.ptrT_ExchgParam^.T_StationCommon.wState:=T_Visu.ptrT_ExchgParam^.T_StationCommon.wState AND 16#BF;
			T_Visu.T_CtrleAction.xDone:=TRUE;
			T_Visu.T_CtrleAction.xNotReady:=FALSE;
			IF (T_Station.THardware.TAxisGrindFeeder.T_Config_Gen.iTyp <> 0) THEN
				diErrorNr:=(T_Station.THardware.TAxisGrindFeeder.T_Config_Gen.iTyp * 1000000) + T_Station.THardware.TAxisGrindFeeder.T_CtrleSingle.udiErrorID;
			ELSE
				diErrorNr:=0;
			END_IF;
			FBErrorMessage(	diErrorNr:=diErrorNr,
							T_ErrorList:=T_ErrorList);
			T_Visu.ptrT_ExchgParam^.T_Visu.T_Message.sDynamicTextEnglish:=FBErrorMessage.sErrorTextEnglish;
			T_Visu.ptrT_ExchgParam^.T_Visu.T_Message.sDynamicTextDeutsch:=FBErrorMessage.sErrorTextDeutsch;
			T_Visu.ptrT_ExchgParam^.T_Visu.T_Message.sDynamicTextFrancais:=FBErrorMessage.sErrorTextFrancais;
			T_Visu.ptrT_ExchgParam^.T_SafetyCtrl.xSetForceError:=TRUE;
			T_Visu.ptrT_ExchgParam^.T_SafetyCtrl.diSetForceErrorNr:=diErrorNr;
			T_Visu.T_CtrleAction.xErr:=FALSE;
			T_Visu.T_CtrleAction.udiErrorID:=0;
			T_Station.THardware.TAxisGrindFeeder.T_CtrleSingle.iFunction:=1;
			T_Station.THardware.TAxisGrindFeeder.T_CtrleSingle.xExecute:=TRUE;
			xOverlayGrindFeedSetPlung:=FALSE;
			T_Visu.ptrT_ExchgParam^.T_FunctionCommon.xOpenOverlaySetGrindPlunge:=FALSE;
			T_Visu.ptrT_ExchgParam^.T_FunctionCommon.xHideProgressbar:=FALSE;
		END_CASE
	END_IF;

(* Plunge On/Off or Displace On/Off *)
	IF xPlungeActivation OR xDisplaceActivation THEN
		CASE iStepAction OF
		(* check visu *)
		1:	xTmp:=	TRUE;
			IF xTmp THEN
				(* next Step *)
				iStepAction :=10;
			(* activ error *)
			ELSE iStepAction:=95; END_IF
		10:	(* Open Overlay *)
			IF xPlungeActivation THEN
				IF (T_Visu.T_PlcParam.dwActualPage = 110) THEN
					T_Visu.ptrT_ExchgParam^.T_StationCommon.T_CalibrationPara.xPlungeActivationCalib:=NOT(T_Visu.ptrT_ExchgParam^.T_StationCommon.T_CalibrationPara.xPlungeActivationCalib);
				ELSIF (T_Visu.T_PlcParam.dwActualPage = 10) THEN
					T_Visu.ptrT_ExchgParam^.T_StationCommon.T_AutoGeometryPara.xPlungeActivationGeometry:=NOT(T_Visu.ptrT_ExchgParam^.T_StationCommon.T_AutoGeometryPara.xPlungeActivationGeometry);
				ELSIF (T_Visu.T_PlcParam.dwActualPage = 20) THEN
					T_Visu.ptrT_ExchgParam^.T_StationCommon.T_AutoGroovePara.xPlungeActivationGroove:=NOT(T_Visu.ptrT_ExchgParam^.T_StationCommon.T_AutoGroovePara.xPlungeActivationGroove);
				END_IF;
			END_IF;
			IF xDisplaceActivation THEN
				IF (T_Visu.T_PlcParam.dwActualPage = 110) THEN
					T_Visu.ptrT_ExchgParam^.T_StationCommon.T_CalibrationPara.xDisplaceActivationCalib:=NOT(T_Visu.ptrT_ExchgParam^.T_StationCommon.T_CalibrationPara.xDisplaceActivationCalib);
				ELSIF (T_Visu.T_PlcParam.dwActualPage = 10) THEN
					T_Visu.ptrT_ExchgParam^.T_StationCommon.T_AutoGeometryPara.xDisplaceActivationGeometry:=NOT(T_Visu.ptrT_ExchgParam^.T_StationCommon.T_AutoGeometryPara.xDisplaceActivationGeometry);
				ELSIF (T_Visu.T_PlcParam.dwActualPage = 20) THEN
					T_Visu.ptrT_ExchgParam^.T_StationCommon.T_AutoGroovePara.xDisplaceActivationGroove:=NOT(T_Visu.ptrT_ExchgParam^.T_StationCommon.T_AutoGroovePara.xDisplaceActivationGroove);
				END_IF;
			END_IF;
			(* next Step *)
			iStepAction :=30;
		(* active saving data NovRAM *)
		30:	xAction_SaveNovRAM:=TRUE;
			iStepActionNovRam:=1;
			(* next step *)
			iStepAction:=40;
		(* waiting confirm saving NovRAM action *)
		40:	IF NOT xAction_SaveNovRAM THEN
				xCalcAgainProcTime:=TRUE;
				iStepAction:=90;
			END_IF;
		(* change page done *)
		90:	T_Visu.T_CtrleAction.xDone:=TRUE;
			T_Visu.T_CtrleAction.xNotReady:=FALSE;
			T_Visu.T_CtrleAction.xErr:=FALSE;
			T_Visu.T_CtrleAction.udiErrorID:=0;
			xPlungeActivation:=FALSE;
			xDisplaceActivation:=FALSE;
		(* not ready *)
		95:	T_Visu.T_CtrleAction.xDone:=TRUE;
			T_Visu.T_CtrleAction.xNotReady:=FALSE;
			T_Visu.T_CtrleAction.xErr:=FALSE;
			T_Visu.T_CtrleAction.udiErrorID:=0;
			xPlungeActivation:=FALSE;
			xDisplaceActivation:=FALSE;
		END_CASE
	END_IF;

(* AutoGroove-->Block GrindFeeder On/Off *)
	IF xBlockGrindFeederActivation THEN
		CASE iStepAction OF
		(* check visu *)
		1:	xTmp:=	TRUE;
			IF xTmp THEN
				(* next Step *)
				iStepAction :=10;
			(* activ error *)
			ELSE iStepAction:=95; END_IF
		10:	(* Open Overlay *)
			T_Visu.ptrT_ExchgParam^.T_StationCommon.T_AutoGroovePara.xBlockGrindFeeder:=NOT(T_Visu.ptrT_ExchgParam^.T_StationCommon.T_AutoGroovePara.xBlockGrindFeeder);
			(* next Step *)
			iStepAction :=30;
		(* active saving data NovRAM *)
		30:	xAction_SaveNovRAM:=TRUE;
			iStepActionNovRam:=1;
			(* next step *)
			iStepAction:=40;
		(* waiting confirm saving NovRAM action *)
		40:	IF NOT xAction_SaveNovRAM THEN
				iStepAction:=90;
			END_IF;
		(* change page done *)
		90:	T_Visu.T_CtrleAction.xDone:=TRUE;
			T_Visu.T_CtrleAction.xNotReady:=FALSE;
			T_Visu.T_CtrleAction.xErr:=FALSE;
			T_Visu.T_CtrleAction.udiErrorID:=0;
			xBlockGrindFeederActivation:=FALSE;
		(* not ready *)
		95:	T_Visu.T_CtrleAction.xDone:=TRUE;
			T_Visu.T_CtrleAction.xNotReady:=FALSE;
			T_Visu.T_CtrleAction.xErr:=FALSE;
			T_Visu.T_CtrleAction.udiErrorID:=0;
			xBlockGrindFeederActivation:=FALSE;
		END_CASE
	END_IF;

(* AutoGroove-->ToolFeeder move to StartPos *)
	IF xToolFeederMoveStartPos OR xToolFeederMoveLoadPos THEN
		(* Step move abs position *)
		CASE iStepAction OF
		(* check axis *)
		1:	IF NOT T_Station.TControl.xHardwareConfigError THEN
				xStepActionDone:=FALSE;
				iStepAction:=95;
				xTmp:=	T_Station.THardware.TAxisToolFeeder.T_CtrleSingle.xDone
						AND T_Station.THardware.TAxisToolFeeder.T_CtrleSingle.xReady
						AND T_Station.THardware.TAxisToolFeeder.T_CtrleSingle.xNotMoving
						AND T_Station.THardware.TAxisToolFeeder.T_CtrleSingle.xPower
						AND NOT(T_Station.THardware.TAxisToolFeeder.T_CtrleSingle.xErr)
						AND NOT(T_Station.THardware.TAxisToolFeeder.T_CtrleSingle.xExecute)
						AND ((T_Station.THardware.TAxisToolFeeder.T_CtrleSingle.xRef AND xMicroRodActive) OR NOT(xMicroRodActive));
				(* Start/Stop position or speed of teachin page has to be confirmed *)
				IF xTmp THEN
					iStepAction:=10;
				ELSE
					IF NOT T_Station.THardware.TAxisToolFeeder.T_CtrleSingle.xRef THEN
					(* Display message, axis not referenced *)
						tTimeOutAction:=TimerAction.ET+T#2s;
						T_Visu.ptrT_ExchgParam^.T_Visu.T_Message.iState:=18;
						(* Action has been cancelled *)
						iStepAction:=89;
					END_IF
				END_IF
			ELSE
				iStepAction:=95;
			END_IF;
		(* activ function axis *)
		10:	tTimeOutAction:=T#999s;
			bStateMachine:=2;
			xSetStateMachine:=TRUE;
			IF xMicroRodActive THEN
				iStepAction:=20;		(* Move Absolut *)
			END_IF;
			IF NOT(xMicroRodActive) THEN
				iStepAction:=35;		(* Move Relativ *)
			END_IF;
			(* init. acc/dec/jerk *)
			T_Station.THardware.TAxisToolFeeder.T_CtrleSingle.lrAcceleration:=T_NovRam.T_Data.T_Standard.T_TeachINToolFeeder.rAcceleration;
			T_Station.THardware.TAxisToolFeeder.T_CtrleSingle.lrDecceleration:=T_NovRam.T_Data.T_Standard.T_TeachINToolFeeder.rDeceleration;
			(*
			T_Station.THardware.TAxisToolFeeder.T_CtrleSingle.lrAcceleration:=T_Station.THardware.TAxisToolFeeder.T_Config_ObjFileValue.lrAcceleration;
			T_Station.THardware.TAxisToolFeeder.T_CtrleSingle.lrDecceleration:=T_Station.THardware.TAxisToolFeeder.T_Config_ObjFileValue.lrDecceleration;
			T_Station.THardware.TAxisToolFeeder.T_CtrleSingle.lrJerk:=T_Station.THardware.TAxisToolFeeder.T_Config_ObjFileValue.lrJerk;
			*)
		(* activ function axis move absolut *)
		20:	IF xToolFeederMoveStartPos THEN
				IF (T_Visu.T_PlcParam.dwActualPage = 10) THEN
					T_Station.THardware.TAxisToolFeeder.T_CtrleSingle.lrPosition:=	T_NovRam.T_Data.T_ProcessImageData.T_ProcessPara.rStartPosToolFeedAuto;
				END_IF;
				IF (T_Visu.T_PlcParam.dwActualPage = 20) THEN
					IF T_NovRam.T_Data.T_ProcessImageData.T_AutoGroovePara.xPlungeActivationGroove AND T_NovRam.T_Data.T_ProcessImageData.T_AutoGroovePara.xBlockGrindFeeder THEN
						T_Station.THardware.TAxisToolFeeder.T_CtrleSingle.lrPosition:=	T_NovRam.T_Data.T_ProcessImageData.T_ProcessPara.rStartPosToolFeedAuto +
																				T_NovRam.T_Data.T_ProcessImageData.T_AutoGroovePara.rPlungeLengthToolFeedGroove;
					ELSE
						T_Station.THardware.TAxisToolFeeder.T_CtrleSingle.lrPosition:=	T_NovRam.T_Data.T_ProcessImageData.T_ProcessPara.rStartPosToolFeedAuto;
					END_IF;
				END_IF;
				IF (T_Visu.T_PlcParam.dwActualPage = 110) THEN
					T_Station.THardware.TAxisToolFeeder.T_CtrleSingle.lrPosition:=	T_NovRam.T_Data.T_ProcessImageData.T_CalibrationPara.rStartPosToolFeedCalib;
				END_IF;
				T_Station.THardware.TAxisToolFeeder.T_CtrleSingle.lrVelocity:=T_NovRam.T_Data.T_ProcessImageData.T_ProcessPara.rSpeedStartPosToolFeedProcess;
			END_IF;
			IF xToolFeederMoveLoadPos THEN
				T_Station.THardware.TAxisToolFeeder.T_CtrleSingle.lrPosition:=	T_NovRam.T_Data.T_Standard.T_AxisPosition.rLoadPosToolFeedAuto;
				T_Station.THardware.TAxisToolFeeder.T_CtrleSingle.lrVelocity:=T_NovRam.T_Data.T_Standard.T_TeachINToolFeeder.rPositionSpeed;
			END_IF;
			T_Station.THardware.TAxisToolFeeder.T_CtrleSingle.iFunction:=7;
			T_Station.THardware.TAxisToolFeeder.T_CtrleSingle.xExecute:=TRUE;
			(* next step *)
			iStepAction:=40;
			xStepActionDone:=FALSE;
		(* activ function axis move relativ *)
		35:	IF (T_Visu.T_PlcParam.dwActualPage = 10) THEN
				T_Station.THardware.TAxisToolFeeder.T_CtrleSingle.lrDistance:=0;
			END_IF;
			IF (T_Visu.T_PlcParam.dwActualPage = 20) THEN
				IF T_NovRam.T_Data.T_ProcessImageData.T_AutoGroovePara.xPlungeActivationGroove (*AND T_NovRam.T_Data.T_ProcessImageData.T_AutoGroovePara.xBlockGrindFeeder*) THEN
					T_Station.THardware.TAxisToolFeeder.T_CtrleSingle.lrDistance:=T_NovRam.T_Data.T_ProcessImageData.T_AutoGroovePara.rPlungeLengthToolFeedGroove;
				ELSE
					(*T_Station.THardware.TAxisToolFeeder.T_CtrleSingle.lrDistance:=0;*)
					iStepAction:=95;
					RETURN;
				END_IF;
			END_IF;
			T_Station.THardware.TAxisToolFeeder.T_CtrleSingle.lrVelocity:=T_NovRam.T_Data.T_ProcessImageData.T_ProcessPara.rSpeedStartPosToolFeedProcess;
			T_Station.THardware.TAxisToolFeeder.T_CtrleSingle.iFunction:=8;
			T_Station.THardware.TAxisToolFeeder.T_CtrleSingle.xExecute:=TRUE;
			(* next step *)
			iStepAction:=40;
			xStepActionDone:=FALSE;
		(* confirm execution *)
		40:	IF NOT(xStepActionDone) THEN
			(* confirm execution *)
				T_Station.THardware.TAxisToolFeeder.T_CtrleSingle.xExecute:=FALSE;
				xStepActionDone:=TRUE;
				(* Display message, 'Start moving' *)
				T_Visu.ptrT_ExchgParam^.T_Visu.T_Message.iState:=26;
			ELSE
				IF T_Station.THardware.TAxisToolFeeder.T_CtrleSingle.xDone THEN
				(* confirm action next step *)
					bStateMachine:=1;
					xSetStateMachine:=TRUE;
					iStepAction:=90;
					xStepActionDone:=FALSE;
				ELSE
					IF T_Station.THardware.TAxisToolFeeder.T_CtrleSingle.xErr THEN
					(* activ action not ready or error *)
						iStepAction:=99;
						xStepActionDone:=FALSE;
					END_IF
				END_IF
			END_IF
		(* waiting timeout *)
		89: IF TimerAction.Q THEN iStepAction:=90; END_IF
			(*T_Visu.ptrT_ExchgParam^.T_TeachIn.iStateAxisMovement:=1;*)
		(* action done *)
		90:	T_Visu.ptrT_ExchgParam^.T_StationCommon.wState:=T_Visu.ptrT_ExchgParam^.T_StationCommon.wState AND 16#BF;
			T_Visu.T_CtrleAction.xDone:=TRUE;
			T_Visu.T_CtrleAction.xNotReady:=FALSE;
			T_Visu.T_CtrleAction.xErr:=FALSE;
			T_Visu.T_CtrleAction.udiErrorID:=0;
			xToolFeederMoveStartPos:=xToolFeederMoveLoadPos:=FALSE;
			(*T_Visu.ptrT_ExchgParam^.T_TeachIn.iStateAxisMovement:=1;*)
		(* axis not ready *)
		95:	T_Visu.ptrT_ExchgParam^.T_StationCommon.wState:=T_Visu.ptrT_ExchgParam^.T_StationCommon.wState AND 16#BF;
			TimerNotReady(IN:=TRUE);
			xToolFeederMoveStartPos:=xToolFeederMoveLoadPos:=FALSE;
			(*T_Visu.ptrT_ExchgParam^.T_TeachIn.iStateAxisMovement:=1;*)
		(* error *)
		99:	T_Visu.ptrT_ExchgParam^.T_StationCommon.wState:=T_Visu.ptrT_ExchgParam^.T_StationCommon.wState AND 16#BF;
			T_Visu.T_CtrleAction.xDone:=TRUE;
			T_Visu.T_CtrleAction.xNotReady:=FALSE;
			IF (T_Station.THardware.TAxisToolFeeder.T_Config_Gen.iTyp <> 0) THEN
				diErrorNr:=(T_Station.THardware.TAxisToolFeeder.T_Config_Gen.iTyp * 1000000) + T_Station.THardware.TAxisToolFeeder.T_CtrleSingle.udiErrorID;
			ELSE
				diErrorNr:=0;
			END_IF;
			FBErrorMessage(	diErrorNr:=diErrorNr,
							T_ErrorList:=T_ErrorList);
			T_Visu.ptrT_ExchgParam^.T_Visu.T_Message.sDynamicTextEnglish:=FBErrorMessage.sErrorTextEnglish;
			T_Visu.ptrT_ExchgParam^.T_Visu.T_Message.sDynamicTextDeutsch:=FBErrorMessage.sErrorTextDeutsch;
			T_Visu.ptrT_ExchgParam^.T_Visu.T_Message.sDynamicTextFrancais:=FBErrorMessage.sErrorTextFrancais;
			T_Visu.ptrT_ExchgParam^.T_SafetyCtrl.xSetForceError:=TRUE;
			T_Visu.ptrT_ExchgParam^.T_SafetyCtrl.diSetForceErrorNr:=diErrorNr;
			T_Visu.T_CtrleAction.xErr:=FALSE;
			T_Visu.T_CtrleAction.udiErrorID:=0;
			T_Station.THardware.TAxisToolFeeder.T_CtrleSingle.iFunction:=1;
			T_Station.THardware.TAxisToolFeeder.T_CtrleSingle.xExecute:=TRUE;
			xToolFeederMoveStartPos:=xToolFeederMoveLoadPos:=FALSE;
			(*T_Visu.ptrT_ExchgParam^.T_TeachIn.iStateAxisMovement:=1;*)
		END_CASE
	END_IF
(*08.07.2014: KFS	{	*)
(* WarmUp On/Off*)
	IF xWarmUp THEN
		CASE iStepAction OF
		(* check visu *)
		1:	xTmp:=	TRUE;
			IF xTmp THEN
				(* next Step *)
				iStepAction :=10;
			(* activ error *)
			ELSE iStepAction:=95; END_IF
		10:	(* Open Overlay *)
			IF (T_Visu.T_PlcParam.dwActualPage = 10) THEN
				T_Visu.ptrT_ExchgParam^.T_StationCommon.T_AutoGeometryPara.xWarmUp:=NOT(T_Visu.ptrT_ExchgParam^.T_StationCommon.T_AutoGeometryPara.xWarmUp);
			END_IF;
			(* next Step *)
			iStepAction :=90;
		(* change page done *)
		90:	T_Visu.T_CtrleAction.xDone:=TRUE;
			T_Visu.T_CtrleAction.xNotReady:=FALSE;
			T_Visu.T_CtrleAction.xErr:=FALSE;
			T_Visu.T_CtrleAction.udiErrorID:=0;
			xWarmUp:=FALSE;
		(* not ready *)
		95:	T_Visu.T_CtrleAction.xDone:=TRUE;
			T_Visu.T_CtrleAction.xNotReady:=FALSE;
			T_Visu.T_CtrleAction.xErr:=FALSE;
			T_Visu.T_CtrleAction.udiErrorID:=0;
			xWarmUp:=FALSE;
		END_CASE
	END_IF;
(*08.07.2014: KFS	}	*)

(*23.02.2023: SOA  {   Reset Warmup if Change of page   *)
IF (T_Visu.T_PlcParam.dwActualPage <> 10) THEN
	T_Visu.ptrT_ExchgParam^.T_StationCommon.T_AutoGeometryPara.xWarmUp := xWarmUp := xWarmUpMessage := xWarmUpMessageActiv := xWarmUpMessageDone := FALSE;
END_IF
(*23.02.2023: SOA  {      *)

